  MoveC 1160 to (433.16, -30.09, -5) mm, rotated rx -180 ry 0 rz -60 deg; joints [3.301, -66.266, 153.274, -56.747, -88.159, 3.391] to (420.46, -17.39, -5) mm, rotated rx 180 ry 0 rz -60 deg; joints [4.068, -65.905, 152.306, -55.999, -87.786, 3.873]
  MoveL 1161 to (395.06, -17.39, -5) mm, rotated rx -180 ry 0 rz -30 deg; joints [13.007, -68.027, 157.856, -16.999, -89.219, 0.721]
  MoveL 1162 to (318.86, -17.39, -5) mm, rotated rx -180 ry 0 rz 0 deg; joints [22.894, -66.084, 152.119, 22.962, -85.478, -1.274]
  MoveC 1163 to (306.16, -30.09, -5) mm, rotated rx 180 ry 0 rz 0 deg; joints [21.838, -65.873, 151.62, 21.912, -85.183, -1.314] to (293.46, -17.39, -5) mm, rotated rx -180 ry 0 rz 0 deg; joints [22.278, -65.412, 150.426, 22.379, -84.518, -1.624]
  MoveL 1164 to (191.86, -17.39, -5) mm, rotated rx -180 ry 0 rz 0 deg; joints [20.102, -62.526, 143.489, 20.378, -80.65, -2.863]
  MoveC 1165 to (179.16, -30.09, -5) mm, rotated rx -180 ry 0 rz 0 deg; joints [19.189, -62.27, 142.918, 19.471, -80.304, -2.833] to (166.46, -17.39, -5) mm, rotated rx -180 ry 0 rz 0 deg; joints [19.62, -61.76, 141.713, 19.95, -79.673, -3.141]
  MoveL 1166 to (90.26, -17.39, -5) mm, rotated rx -180 ry 0 rz 0 deg; joints [18.3, -59.367, 136.274, 18.815, -76.713, -3.918]
  MoveL 1167 to (64.86, -17.39, -5) mm, rotated rx -180 ry 0 rz 0 deg; joints [17.897, -58.538, 134.424, 18.482, -75.714, -4.162]
  MoveC 1168 to (61.14, -26.37, -5) mm, rotated rx -180 ry 0 rz 0 deg; joints [17.408, -58.504, 134.36, 17.981, -75.65, -4.054] to (52.16, -30.09, -5) mm, rotated rx -180 ry 0 rz 0 deg; joints [17.095, -58.242, 133.784, 17.684, -75.327, -4.078]
  MoveL 1169 to (52.16, -30.09, -5) mm, rotated rx -180 ry 0 rz 0 deg; joints [17.095, -58.242, 133.784, 17.684, -75.327, -4.078]
  MoveC 1170 to (43.18, -26.37, -5) mm, rotated rx -180 ry 0 rz 0 deg; joints [17.141, -57.907, 133.035, 17.765, -74.936, -4.219] to (39.46, -17.39, -5) mm, rotated rx -180 ry 0 rz 0 deg; joints [17.511, -57.695, 132.553, 18.169, -74.709, -4.4]
  MoveL 1171 to (14.06, -17.39, -5) mm, rotated rx -180 ry 0 rz 0 deg; joints [17.141, -56.836, 130.661, 17.877, -73.696, -4.634]
  MoveC 1172 to (13.61, -17.2, -5) mm, rotated rx -180 ry 0 rz 0 deg; joints [17.143, -56.818, 130.623, 17.881, -73.676, -4.641] to (13.42, -16.75, -5) mm, rotated rx -180 ry 0 rz 0 deg; joints [17.161, -56.808, 130.599, 17.901, -73.665, -4.65]
  MoveL 1173 to (13.42, -16.12, -5) mm, rotated rx 180 ry 0 rz 0 deg; joints [17.191, -56.801, 130.584, 17.932, -73.659, -4.661]
  MoveC 1174 to (13.42, -15.67, -4.81) mm, rotated rx -180 ry 0 rz 0 deg; joints [17.211, -56.81, 130.574, 17.955, -73.643, -4.673] to (13.42, -15.48, -4.37) mm, rotated rx -180 ry 0 rz 0 deg; joints [17.22, -56.839, 130.571, 17.967, -73.613, -4.686]
  Set speed (500.0 mm/s)
  MoveL 1175 to (13.42, -15.48, 5) mm, rotated rx -180 ry 0 rz 0 deg; joints [17.216, -57.49, 130.588, 18.021, -73.01, -4.889]
  MoveL 1176 to (12.15, -16.75, 5) mm, rotated rx 180 ry 0 rz 0 deg; joints [17.139, -57.459, 130.522, 17.945, -72.97, -4.878]
  Set speed (25.4 mm/s)
  MoveL 1177 to (12.15, -16.75, 1) mm, rotated rx -180 ry 0 rz 0 deg; joints [17.141, -57.181, 130.516, 17.921, -73.228, -4.791]
  MoveL 1178 to (12.15, -16.75, -7.72) mm, rotated rx 180 ry 0 rz 0 deg; joints [17.144, -56.575, 130.497, 17.871, -73.788, -4.604]
  MoveC 1179 to (12.34, -16.75, -8.16) mm, rotated rx -180 ry 0 rz 0 deg; joints [17.147, -56.55, 130.51, 17.871, -73.824, -4.592] to (12.79, -16.75, -8.35) mm, rotated rx 180 ry 0 rz 0 deg; joints [17.154, -56.552, 130.543, 17.875, -73.854, -4.584]
  Set speed (50.8 mm/s)
  MoveL 1180 to (13.42, -16.75, -8.35) mm, rotated rx -180 ry 0 rz 0 deg; joints [17.163, -56.574, 130.591, 17.882, -73.88, -4.578]
  MoveC 1181 to (13.87, -16.94, -8.35) mm, rotated rx -180 ry 0 rz 0 deg; joints [17.161, -56.591, 130.628, 17.878, -73.899, -4.571] to (14.06, -17.39, -8.35) mm, rotated rx -180 ry 0 rz 0 deg; joints [17.143, -56.601, 130.653, 17.858, -73.911, -4.562]
  MoveL 1182 to (14.06, -169.79, -8.35) mm, rotated rx -180 ry 0 rz 0 deg; joints [9.848, -57.754, 133.422, 10.193, -75.015, -2.239]
  MoveL 1183 to (471.26, -169.79, -8.35) mm, rotated rx -180 ry 0 rz -60 deg; joints [-6.049, -66.719, 155.749, -66.059, -89.408, 1.775]
  MoveL 1184 to (471.26, -17.39, -8.35) mm, rotated rx 180 ry 0 rz -60 deg; joints [4.314, -66.857, 155.917, -55.696, -89.272, 1.665]
  MoveL 1185 to (445.86, -17.39, -8.35) mm, rotated rx -180 ry 0 rz -60 deg; joints [4.188, -66.217, 154.11, -55.84, -88.618, 2.632]
  MoveC 1186 to (433.16, -30.09, -8.35) mm, rotated rx -180 ry 0 rz -60 deg; joints [3.303, -65.899, 153.262, -56.737, -88.354, 3.094] to (420.46, -17.39, -8.35) mm, rotated rx 180 ry 0 rz -60 deg; joints [4.069, -65.548, 152.294, -55.987, -87.979, 3.586]
  MoveL 1187 to (395.06, -17.39, -8.35) mm, rotated rx 180 ry 0 rz -30 deg; joints [13.009, -67.611, 157.843, -16.996, -89.605, 0.603]
  MoveL 1188 to (318.86, -17.39, -8.35) mm, rotated rx 180 ry 0 rz 0 deg; joints [22.896, -65.729, 152.107, 22.954, -85.795, -1.139]
  MoveC 1189 to (306.16, -30.09, -8.35) mm, rotated rx -180 ry 0 rz 0 deg; joints [21.84, -65.522, 151.609, 21.904, -85.499, -1.187] to (293.46, -17.39, -8.35) mm, rotated rx -180 ry 0 rz 0 deg; joints [22.28, -65.07, 150.415, 22.369, -84.823, -1.498]
  MoveL 1190 to (191.86, -17.39, -8.35) mm, rotated rx -180 ry 0 rz 0 deg; joints [20.104, -62.233, 143.48, 20.364, -80.916, -2.763]
  MoveC 1191 to (179.16, -30.09, -8.35) mm, rotated rx 180 ry 0 rz 0 deg; joints [19.19, -61.98, 142.909, 19.457, -80.568, -2.738] to (166.46, -17.39, -8.35) mm, rotated rx -180 ry 0 rz 0 deg; joints [19.622, -61.477, 141.703, 19.935, -79.93, -3.046]
  MoveL 1192 to (90.26, -17.39, -8.35) mm, rotated rx -180 ry 0 rz 0 deg; joints [18.302, -59.111, 136.266, 18.798, -76.947, -3.836]
  MoveL 1193 to (64.86, -17.39, -8.35) mm, rotated rx -180 ry 0 rz 0 deg; joints [17.899, -58.29, 134.415, 18.465, -75.942, -4.084]
  MoveC 1194 to (61.14, -26.37, -8.35) mm, rotated rx -180 ry 0 rz 0 deg; joints [17.41, -58.255, 134.351, 17.964, -75.878, -3.978] to (52.16, -30.09, -8.35) mm, rotated rx -180 ry 0 rz 0 deg; joints [17.097, -57.996, 133.775, 17.667, -75.553, -4.004]
  MoveL 1195 to (52.16, -30.09, -8.35) mm, rotated rx -180 ry 0 rz 0 deg; joints [17.097, -57.996, 133.775, 17.667, -75.553, -4.004]
  MoveC 1196 to (43.18, -26.37, -8.35) mm, rotated rx -180 ry 0 rz 0 deg; joints [17.142, -57.664, 133.027, 17.747, -75.16, -4.146] to (39.46, -17.39, -8.35) mm, rotated rx -180 ry 0 rz 0 deg; joints [17.513, -57.453, 132.544, 18.151, -74.93, -4.325]
  MoveL 1197 to (14.06, -17.39, -8.35) mm, rotated rx -180 ry 0 rz 0 deg; joints [17.143, -56.601, 130.653, 17.858, -73.911, -4.562]
  MoveC 1198 to (13.61, -17.2, -8.35) mm, rotated rx -180 ry 0 rz 0 deg; joints [17.145, -56.584, 130.615, 17.862, -73.891, -4.569] to (13.42, -16.75, -8.35) mm, rotated rx -180 ry 0 rz 0 deg; joints [17.163, -56.574, 130.591, 17.882, -73.88, -4.578]
  MoveL 1199 to (13.42, -16.12, -8.35) mm, rotated rx -180 ry 0 rz 0 deg; joints [17.192, -56.567, 130.576, 17.913, -73.874, -4.589]
  MoveC 1200 to (13.42, -15.67, -8.16) mm, rotated rx -180 ry 0 rz 0 deg; joints [17.213, -56.576, 130.566, 17.936, -73.858, -4.601] to (13.42, -15.48, -7.72) mm, rotated rx -180 ry 0 rz 0 deg; joints [17.221, -56.606, 130.563, 17.948, -73.828, -4.613]
  Set speed (500.0 mm/s)
  MoveL 1201 to (13.42, -15.48, 6) mm, rotated rx -180 ry 0 rz 0 deg; joints [17.215, -57.56, 130.589, 18.027, -72.945, -4.911]
  MoveL 1202 to (-18.41, -15.48, 6) mm, rotated rx -180 ry 0 rz 0 deg; joints [16.771, -56.434, 128.187, 17.688, -71.688, -5.187]
  Set speed (25.4 mm/s)
  MoveL 1203 to (-18.41, -15.48, -4.37) mm, rotated rx -180 ry 0 rz 0 deg; joints [16.775, -55.739, 128.169, 17.626, -72.334, -4.973]
  MoveC 1204 to (-18.41, -15.67, -4.81) mm, rotated rx 180 ry 0 rz 0 deg; joints [16.767, -55.711, 128.173, 17.614, -72.363, -4.96] to (-18.41, -16.12, -5) mm, rotated rx -180 ry 0 rz 0 deg; joints [16.747, -55.703, 128.182, 17.591, -72.379, -4.948]
  Set speed (50.8 mm/s)
  MoveL 1205 to (-18.41, -16.75, -5) mm, rotated rx -180 ry 0 rz 0 deg; joints [16.718, -55.709, 128.197, 17.56, -72.384, -4.937]
  MoveC 1206 to (-18.6, -17.2, -5) mm, rotated rx 180 ry 0 rz 0 deg; joints [16.695, -55.707, 128.193, 17.537, -72.38, -4.931] to (-19.04, -17.39, -5) mm, rotated rx -180 ry 0 rz 0 deg; joints [16.681, -55.693, 128.163, 17.523, -72.364, -4.932]
  MoveL 1207 to (-39.46, -17.39, -5) mm, rotated rx -180 ry 0 rz 0 deg; joints [16.409, -54.976, 126.603, 17.321, -71.535, -5.113]
  MoveC 1208 to (-52.16, -30.09, -5) mm, rotated rx -180 ry 0 rz 0 deg; joints [15.682, -54.647, 125.906, 16.593, -71.115, -4.993] to (-64.86, -17.39, -5) mm, rotated rx -180 ry 0 rz 0 deg; joints [16.082, -54.069, 124.641, 17.084, -70.495, -5.336]
  MoveL 1209 to (-90.26, -17.39, -5) mm, rotated rx -180 ry 0 rz 0 deg; joints [15.768, -53.146, 122.653, 16.865, -69.445, -5.558]
  MoveL 1210 to (-166.46, -17.39, -5) mm, rotated rx 180 ry 0 rz 0 deg; joints [14.894, -50.279, 116.527, 16.305, -66.228, -6.221]
  MoveC 1211 to (-179.16, -30.09, -5) mm, rotated rx -180 ry 0 rz 0 deg; joints [14.242, -49.907, 115.751, 15.645, -65.767, -6.064] to (-191.86, -17.39, -5) mm, rotated rx -180 ry 0 rz 0 deg; joints [14.623, -49.288, 114.425, 16.15, -65.13, -6.444]
  MoveL 1212 to (-293.46, -17.39, -5) mm, rotated rx -180 ry 0 rz 0 deg; joints [13.63, -45.126, 105.665, 15.689, -60.583, -7.372]
  MoveC 1213 to (-306.16, -30.09, -5) mm, rotated rx -180 ry 0 rz 0 deg; joints [13.04, -44.706, 104.795, 15.083, -60.073, -7.184] to (-318.86, -17.39, -5) mm, rotated rx -180 ry 0 rz 0 deg; joints [13.402, -44.031, 103.374, 15.614, -59.402, -7.617]
  MoveL 1214 to (-395.06, -17.39, -5) mm, rotated rx -180 ry 0 rz 0 deg; joints [12.761, -40.591, 96.21, 15.497, -55.722, -8.407]
  MoveL 1215 to (-420.46, -17.39, -5) mm, rotated rx 180 ry 0 rz 0 deg; joints [12.56, -39.385, 93.71, 15.497, -54.444, -8.693]
  MoveC 1216 to (-433.16, -30.09, -5) mm, rotated rx 180 ry 0 rz 0 deg; joints [12.022, -38.9, 92.714, 14.938, -53.869, -8.482] to (-445.86, -17.39, -5) mm, rotated rx -180 ry 0 rz 0 deg; joints [12.366, -38.146, 91.146, 15.519, -53.136, -8.995]
  MoveL 1217 to (-471.26, -17.39, -5) mm, rotated rx -180 ry 0 rz 0 deg; joints [12.178, -36.871, 88.511, 15.564, -51.795, -9.314]
  MoveL 1218 to (-471.26, -169.79, -5) mm, rotated rx -180 ry 0 rz 0 deg; joints [6.925, -38.12, 91.194, 8.733, -52.522, -4.962]
  MoveL 1219 to (-14.06, -169.79, -5) mm, rotated rx -180 ry 0 rz 0 deg; joints [9.613, -57.027, 131.277, 10.019, -73.608, -2.435]
  MoveL 1220 to (-14.06, -17.39, -5) mm, rotated rx 180 ry 0 rz 0 deg; joints [16.749, -55.867, 128.542, 17.574, -72.565, -4.887]
  MoveL 1221 to (-19.04, -17.39, -5) mm, rotated rx -180 ry 0 rz 0 deg; joints [16.681, -55.693, 128.163, 17.523, -72.364, -4.932]
  MoveC 1222 to (-19.49, -17.2, -5) mm, rotated rx -180 ry 0 rz 0 deg; joints [16.683, -55.676, 128.125, 17.528, -72.344, -4.939] to (-19.68, -16.75, -5) mm, rotated rx -180 ry 0 rz 0 deg; joints [16.701, -55.665, 128.1, 17.547, -72.333, -4.949]
  MoveL 1223 to (-19.68, -16.12, -5) mm, rotated rx -180 ry 0 rz 0 deg; joints [16.73, -55.659, 128.086, 17.578, -72.327, -4.96]
  MoveC 1224 to (-19.68, -15.67, -4.81) mm, rotated rx -180 ry 0 rz 0 deg; joints [16.75, -55.667, 128.076, 17.601, -72.312, -4.972] to (-19.68, -15.48, -4.37) mm, rotated rx 180 ry 0 rz 0 deg; joints [16.758, -55.695, 128.073, 17.613, -72.283, -4.984]
  Set speed (500.0 mm/s)
  MoveL 1225 to (-19.68, -15.48, 5) mm, rotated rx 180 ry 0 rz 0 deg; joints [16.754, -56.322, 128.089, 17.669, -71.7, -5.178]
  MoveL 1226 to (-18.41, -15.48, 5) mm, rotated rx -180 ry 0 rz 0 deg; joints [16.771, -56.368, 128.186, 17.682, -71.751, -5.167]
  Set speed (25.4 mm/s)
  MoveL 1227 to (-18.41, -15.48, 1) mm, rotated rx -180 ry 0 rz 0 deg; joints [16.773, -56.1, 128.18, 17.657, -72.001, -5.083]
  MoveL 1228 to (-18.41, -15.48, -7.72) mm, rotated rx -180 ry 0 rz 0 deg; joints [16.777, -55.514, 128.161, 17.606, -72.542, -4.904]
  MoveC 1229 to (-18.41, -15.67, -8.16) mm, rotated rx -180 ry 0 rz 0 deg; joints [16.769, -55.485, 128.164, 17.595, -72.571, -4.892] to (-18.41, -16.12, -8.35) mm, rotated rx -180 ry 0 rz 0 deg; joints [16.748, -55.477, 128.174, 17.572, -72.586, -4.88]
  Set speed (50.8 mm/s)
  MoveL 1230 to (-18.41, -16.75, -8.35) mm, rotated rx -180 ry 0 rz 0 deg; joints [16.72, -55.483, 128.189, 17.541, -72.592, -4.869]
  MoveC 1231 to (-18.6, -17.2, -8.35) mm, rotated rx 180 ry 0 rz 0 deg; joints [16.697, -55.481, 128.185, 17.518, -72.588, -4.863] to (-19.04, -17.39, -8.35) mm, rotated rx -180 ry 0 rz 0 deg; joints [16.682, -55.468, 128.155, 17.504, -72.571, -4.863]
  MoveL 1232 to (-39.46, -17.39, -8.35) mm, rotated rx 180 ry 0 rz 0 deg; joints [16.41, -54.755, 126.595, 17.301, -71.738, -5.047]
  MoveC 1233 to (-52.16, -30.09, -8.35) mm, rotated rx -180 ry 0 rz 0 deg; joints [15.683, -54.428, 125.898, 16.574, -71.317, -4.929] to (-64.86, -17.39, -8.35) mm, rotated rx -180 ry 0 rz 0 deg; joints [16.084, -53.854, 124.633, 17.064, -70.693, -5.272]
  MoveL 1234 to (-90.26, -17.39, -8.35) mm, rotated rx -180 ry 0 rz 0 deg; joints [15.769, -52.937, 122.646, 16.844, -69.638, -5.496]
  MoveL 1235 to (-166.46, -17.39, -8.35) mm, rotated rx -180 ry 0 rz 0 deg; joints [14.895, -50.085, 116.519, 16.283, -66.407, -6.165]
  MoveC 1236 to (-179.16, -30.09, -8.35) mm, rotated rx 180 ry 0 rz 0 deg; joints [14.243, -49.715, 115.744, 15.624, -65.945, -6.01] to (-191.86, -17.39, -8.35) mm, rotated rx -180 ry 0 rz 0 deg; joints [14.624, -49.098, 114.417, 16.128, -65.305, -6.389]
  MoveL 1237 to (-293.46, -17.39, -8.35) mm, rotated rx 180 ry 0 rz 0 deg; joints [13.631, -44.953, 105.657, 15.665, -60.743, -7.321]
  MoveC 1238 to (-306.16, -30.09, -8.35) mm, rotated rx -180 ry 0 rz 0 deg; joints [13.041, -44.534, 104.788, 15.06, -60.232, -7.135] to (-318.86, -17.39, -8.35) mm, rotated rx -180 ry 0 rz 0 deg; joints [13.403, -43.862, 103.367, 15.59, -59.558, -7.567]
  MoveL 1239 to (-395.06, -17.39, -8.35) mm, rotated rx -180 ry 0 rz 0 deg; joints [12.762, -40.431, 96.203, 15.471, -55.869, -8.358]
  MoveL 1240 to (-420.46, -17.39, -8.35) mm, rotated rx 180 ry 0 rz 0 deg; joints [12.561, -39.229, 93.703, 15.47, -54.588, -8.645]
  MoveC 1241 to (-433.16, -30.09, -8.35) mm, rotated rx -180 ry 0 rz 0 deg; joints [12.023, -38.744, 92.707, 14.911, -54.012, -8.436] to (-445.86, -17.39, -8.35) mm, rotated rx -180 ry 0 rz 0 deg; joints [12.367, -37.993, 91.139, 15.491, -53.277, -8.947]
  MoveL 1242 to (-471.26, -17.39, -8.35) mm, rotated rx 180 ry 0 rz 0 deg; joints [12.178, -36.721, 88.504, 15.535, -51.933, -9.266]
  MoveL 1243 to (-471.26, -169.79, -8.35) mm, rotated rx 180 ry 0 rz 0 deg; joints [6.926, -37.966, 91.187, 8.717, -52.667, -4.934]
  MoveL 1244 to (-14.06, -169.79, -8.35) mm, rotated rx -180 ry 0 rz 0 deg; joints [9.614, -56.791, 131.269, 10.008, -73.832, -2.394]
  MoveL 1245 to (-14.06, -17.39, -8.35) mm, rotated rx -180 ry 0 rz 0 deg; joints [16.75, -55.64, 128.534, 17.555, -72.774, -4.818]
  MoveL 1246 to (-19.04, -17.39, -8.35) mm, rotated rx -180 ry 0 rz 0 deg; joints [16.682, -55.468, 128.155, 17.504, -72.571, -4.863]
  MoveC 1247 to (-19.49, -17.2, -8.35) mm, rotated rx -180 ry 0 rz 0 deg; joints [16.685, -55.45, 128.117, 17.508, -72.551, -4.871] to (-19.68, -16.75, -8.35) mm, rotated rx -180 ry 0 rz 0 deg; joints [16.702, -55.439, 128.092, 17.528, -72.54, -4.88]
  MoveL 1248 to (-19.68, -16.12, -8.35) mm, rotated rx -180 ry 0 rz 0 deg; joints [16.731, -55.433, 128.078, 17.559, -72.535, -4.891]
  MoveC 1249 to (-19.68, -15.67, -8.16) mm, rotated rx -180 ry 0 rz 0 deg; joints [16.751, -55.441, 128.068, 17.582, -72.519, -4.903] to (-19.68, -15.48, -7.72) mm, rotated rx -180 ry 0 rz 0 deg; joints [16.76, -55.47, 128.065, 17.593, -72.49, -4.916]
  Set speed (500.0 mm/s)
  MoveL 1250 to (-19.68, -15.48, 6) mm, rotated rx 180 ry 0 rz 0 deg; joints [16.754, -56.389, 128.091, 17.675, -71.638, -5.198]
  MoveL 1251 to (-13.42, -196.52, 6) mm, rotated rx 180 ry 0 rz 0 deg; joints [8.324, -57.961, 131.671, 8.701, -73.018, -2.16]
  Set speed (25.4 mm/s)
  MoveL 1252 to (-13.42, -196.51, -4.36) mm, rotated rx -180 ry 0 rz 0 deg; joints [8.327, -57.228, 131.652, 8.672, -73.724, -2.048]
  MoveC 1253 to (-13.42, -196.7, -4.81) mm, rotated rx -180 ry 0 rz 0 deg; joints [8.318, -57.197, 131.653, 8.661, -73.755, -2.041] to (-13.42, -197.15, -5) mm, rotated rx 180 ry 0 rz 0 deg; joints [8.297, -57.186, 131.658, 8.638, -73.77, -2.032]
  Set speed (50.8 mm/s)
  MoveL 1254 to (-13.42, -197.79, -5) mm, rotated rx 180 ry 0 rz 0 deg; joints [8.266, -57.189, 131.665, 8.606, -73.773, -2.023]
  MoveC 1255 to (-13.61, -198.23, -5) mm, rotated rx -180 ry 0 rz 0 deg; joints [8.243, -57.184, 131.656, 8.582, -73.767, -2.018] to (-14.06, -198.42, -5) mm, rotated rx -180 ry 0 rz 0 deg; joints [8.23, -57.17, 131.623, 8.57, -73.749, -2.017]
  MoveL 1256 to (-39.46, -198.42, -5) mm, rotated rx 180 ry 0 rz 0 deg; joints [8.056, -56.276, 129.652, 8.437, -72.676, -2.133]
  MoveC 1257 to (-52.16, -211.12, -5) mm, rotated rx -180 ry 0 rz 0 deg; joints [7.375, -55.879, 128.793, 7.743, -72.191, -1.996] to (-64.86, -198.42, -5) mm, rotated rx -180 ry 0 rz 0 deg; joints [7.889, -55.367, 127.661, 8.312, -71.598, -2.248]
  MoveL 1258 to (-90.26, -198.42, -5) mm, rotated rx -180 ry 0 rz 0 deg; joints [7.729, -54.442, 125.647, 8.197, -70.513, -2.361]
  MoveL 1259 to (-166.46, -198.42, -5) mm, rotated rx -180 ry 0 rz 0 deg; joints [7.285, -51.573, 119.46, 7.9, -67.207, -2.694]
  MoveC 1260 to (-179.16, -211.12, -5) mm, rotated rx 180 ry 0 rz 0 deg; joints [6.674, -51.136, 118.535, 7.265, -66.692, -2.514] to (-191.86, -198.42, -5) mm, rotated rx -180 ry 0 rz 0 deg; joints [7.148, -50.583, 117.344, 7.818, -66.084, -2.805]
  MoveL 1261 to (-293.46, -198.42, -5) mm, rotated rx -180 ry 0 rz 0 deg; joints [6.648, -46.437, 108.562, 7.567, -61.46, -3.258]
  MoveC 1262 to (-306.16, -211.12, -5) mm, rotated rx 180 ry 0 rz 0 deg; joints [6.095, -45.951, 107.55, 6.973, -60.905, -3.039] to (-318.86, -198.42, -5) mm, rotated rx 180 ry 0 rz 0 deg; joints [6.534, -45.349, 106.274, 7.524, -60.264, -3.376]
  MoveL 1263 to (-395.06, -198.42, -5) mm, rotated rx -180 ry 0 rz 0 deg; joints [6.213, -41.939, 99.145, 7.446, -56.555, -3.753]
  MoveL 1264 to (-420.46, -198.42, -5) mm, rotated rx -180 ry 0 rz 0 deg; joints [6.113, -40.749, 96.667, 7.439, -55.271, -3.889]
  MoveC 1265 to (-433.16, -211.12, -5) mm, rotated rx 180 ry 0 rz 0 deg; joints [5.608, -40.201, 95.535, 6.874, -54.656, -3.632] to (-445.86, -198.42, -5) mm, rotated rx -180 ry 0 rz 0 deg; joints [6.016, -39.527, 94.13, 7.441, -53.959, -4.031]
  MoveL 1266 to (-471.26, -198.42, -5) mm, rotated rx 180 ry 0 rz 0 deg; joints [5.922, -38.273, 91.528, 7.455, -52.616, -4.18]
  MoveL 1267 to (-471.26, -350.82, -5) mm, rotated rx 180 ry 0 rz 0 deg; joints [0.538, -38.663, 92.418, 0.669, -52.887, -0.124]
  MoveL 1268 to (-14.06, -350.82, -5) mm, rotated rx 180 ry 0 rz 0 deg; joints [0.749, -57.524, 132.551, 0.774, -74.159, 0.072]
  MoveL 1269 to (-14.06, -198.42, -5) mm, rotated rx -180 ry 0 rz 0 deg; joints [8.23, -57.17, 131.623, 8.57, -73.749, -2.017]
  MoveC 1270 to (-13.87, -197.97, -5) mm, rotated rx 180 ry 0 rz 0 deg; joints [8.254, -57.174, 131.633, 8.594, -73.755, -2.023] to (-13.42, -197.79, -5) mm, rotated rx 180 ry 0 rz 0 deg; joints [8.266, -57.189, 131.665, 8.606, -73.773, -2.023]
  MoveL 1271 to (-12.79, -197.79, -5) mm, rotated rx 180 ry 0 rz 0 deg; joints [8.27, -57.211, 131.714, 8.609, -73.799, -2.02]
  MoveC 1272 to (-12.34, -197.79, -4.81) mm, rotated rx 180 ry 0 rz 0 deg; joints [8.273, -57.24, 131.749, 8.612, -73.806, -2.02] to (-12.15, -197.78, -4.37) mm, rotated rx -180 ry 0 rz 0 deg; joints [8.274, -57.278, 131.765, 8.615, -73.783, -2.024]
  Set speed (500.0 mm/s)
  MoveL 1273 to (-12.15, -197.79, 5) mm, rotated rx 180 ry 0 rz 0 deg; joints [8.271, -57.941, 131.782, 8.64, -73.145, -2.124]
  MoveL 1274 to (-13.42, -196.52, 5) mm, rotated rx 180 ry 0 rz 0 deg; joints [8.324, -57.89, 131.67, 8.698, -73.087, -2.149]
  Set speed (25.4 mm/s)
  MoveL 1275 to (-13.42, -196.51, 1) mm, rotated rx 180 ry 0 rz 0 deg; joints [8.325, -57.608, 131.664, 8.687, -73.359, -2.106]
  MoveL 1276 to (-13.42, -196.52, -7.72) mm, rotated rx -180 ry 0 rz 0 deg; joints [8.328, -56.99, 131.644, 8.663, -73.951, -2.013]
  MoveC 1277 to (-13.42, -196.7, -8.16) mm, rotated rx 180 ry 0 rz 0 deg; joints [8.319, -56.959, 131.645, 8.653, -73.982, -2.005] to (-13.42, -197.15, -8.35) mm, rotated rx -180 ry 0 rz 0 deg; joints [8.298, -56.948, 131.65, 8.629, -73.996, -1.997]
  Set speed (50.8 mm/s)
  MoveL 1278 to (-13.42, -197.79, -8.35) mm, rotated rx -180 ry 0 rz 0 deg; joints [8.267, -56.951, 131.657, 8.597, -73.999, -1.988]
  MoveC 1279 to (-13.61, -198.23, -8.35) mm, rotated rx 180 ry 0 rz 0 deg; joints [8.244, -56.947, 131.647, 8.573, -73.994, -1.982] to (-14.06, -198.42, -8.35) mm, rotated rx -180 ry 0 rz 0 deg; joints [8.232, -56.932, 131.615, 8.562, -73.975, -1.982]
  MoveL 1280 to (-39.46, -198.42, -8.35) mm, rotated rx 180 ry 0 rz 0 deg; joints [8.057, -56.045, 129.644, 8.428, -72.896, -2.1]
  MoveC 1281 to (-52.16, -211.12, -8.35) mm, rotated rx -180 ry 0 rz 0 deg; joints [7.376, -55.651, 128.785, 7.734, -72.409, -1.966] to (-64.86, -198.42, -8.35) mm, rotated rx -180 ry 0 rz 0 deg; joints [7.89, -55.143, 127.653, 8.303, -71.812, -2.215]
  MoveL 1282 to (-90.26, -198.42, -8.35) mm, rotated rx -180 ry 0 rz 0 deg; joints [7.73, -54.224, 125.639, 8.187, -70.721, -2.329]
  MoveL 1283 to (-166.46, -198.42, -8.35) mm, rotated rx -180 ry 0 rz 0 deg; joints [7.286, -51.372, 119.453, 7.89, -67.398, -2.665]
  MoveC 1284 to (-179.16, -211.12, -8.35) mm, rotated rx -180 ry 0 rz 0 deg; joints [6.675, -50.937, 118.527, 7.255, -66.882, -2.488] to (-191.86, -198.42, -8.35) mm, rotated rx 180 ry 0 rz 0 deg; joints [7.149, -50.387, 117.337, 7.808, -66.271, -2.777]
  MoveL 1285 to (-293.46, -198.42, -8.35) mm, rotated rx 180 ry 0 rz 0 deg; joints [6.649, -46.258, 108.554, 7.556, -61.63, -3.233]
  MoveC 1286 to (-306.16, -211.12, -8.35) mm, rotated rx 180 ry 0 rz 0 deg; joints [6.095, -45.775, 107.542, 6.963, -61.073, -3.016] to (-318.86, -198.42, -8.35) mm, rotated rx -180 ry 0 rz 0 deg; joints [6.534, -45.174, 106.267, 7.513, -60.43, -3.352]
  MoveL 1287 to (-395.06, -198.42, -8.35) mm, rotated rx -180 ry 0 rz 0 deg; joints [6.214, -41.776, 99.138, 7.434, -56.71, -3.73]
  MoveL 1288 to (-420.46, -198.42, -8.35) mm, rotated rx -180 ry 0 rz 0 deg; joints [6.114, -40.588, 96.659, 7.426, -55.422, -3.865]
  MoveC 1289 to (-433.16, -211.12, -8.35) mm, rotated rx -180 ry 0 rz 0 deg; joints [5.608, -40.042, 95.528, 6.862, -54.807, -3.61] to (-445.86, -198.42, -8.35) mm, rotated rx -180 ry 0 rz 0 deg; joints [6.017, -39.37, 94.122, 7.428, -54.107, -4.007]
  MoveL 1290 to (-471.26, -198.42, -8.35) mm, rotated rx -180 ry 0 rz 0 deg; joints [5.923, -38.119, 91.521, 7.441, -52.762, -4.157]
  MoveL 1291 to (-471.26, -350.82, -8.35) mm, rotated rx -180 ry 0 rz 0 deg; joints [0.539, -38.508, 92.411, 0.669, -53.035, -0.122]
  MoveL 1292 to (-14.06, -350.82, -8.35) mm, rotated rx -180 ry 0 rz 0 deg; joints [0.75, -57.282, 132.542, 0.774, -74.391, 0.075]
  MoveL 1293 to (-14.06, -198.42, -8.35) mm, rotated rx -180 ry 0 rz 0 deg; joints [8.232, -56.932, 131.615, 8.562, -73.975, -1.982]
  MoveC 1294 to (-13.87, -197.97, -8.35) mm, rotated rx 180 ry 0 rz 0 deg; joints [8.255, -56.936, 131.624, 8.585, -73.981, -1.987] to (-13.42, -197.79, -8.35) mm, rotated rx -180 ry 0 rz 0 deg; joints [8.267, -56.951, 131.657, 8.597, -73.999, -1.988]
  MoveL 1295 to (-12.79, -197.78, -8.35) mm, rotated rx -180 ry 0 rz 0 deg; joints [8.271, -56.973, 131.706, 8.601, -74.026, -1.985]
  MoveC 1296 to (-12.34, -197.78, -8.16) mm, rotated rx 180 ry 0 rz 0 deg; joints [8.274, -57.002, 131.741, 8.604, -74.033, -1.985] to (-12.15, -197.79, -7.72) mm, rotated rx -180 ry 0 rz 0 deg; joints [8.276, -57.04, 131.756, 8.606, -74.01, -1.988]
  Set speed (500.0 mm/s)
  MoveL 1297 to (-12.15, -197.79, 6) mm, rotated rx 180 ry 0 rz 0 deg; joints [8.271, -58.012, 131.784, 8.643, -73.076, -2.135]
  MoveL 1298 to (12.15, -197.78, 6) mm, rotated rx -180 ry 0 rz 0 deg; joints [8.446, -58.875, 133.65, 8.78, -74.075, -2.025]
  Set speed (25.4 mm/s)
  MoveL 1299 to (12.15, -197.79, -4.36) mm, rotated rx 180 ry 0 rz 0 deg; joints [8.449, -58.119, 133.631, 8.753, -74.803, -1.91]
  MoveC 1300 to (12.34, -197.79, -4.81) mm, rotated rx -180 ry 0 rz 0 deg; joints [8.451, -58.093, 133.644, 8.753, -74.842, -1.904] to (12.79, -197.78, -5) mm, rotated rx -180 ry 0 rz 0 deg; joints [8.454, -58.095, 133.677, 8.755, -74.874, -1.9]
  Set speed (50.8 mm/s)
  MoveL 1301 to (13.42, -197.78, -5) mm, rotated rx -180 ry 0 rz 0 deg; joints [8.459, -58.117, 133.726, 8.759, -74.9, -1.897]
  MoveC 1302 to (13.87, -197.97, -5) mm, rotated rx -180 ry 0 rz 0 deg; joints [8.453, -58.133, 133.762, 8.752, -74.92, -1.892] to (14.06, -198.42, -5) mm, rotated rx -180 ry 0 rz 0 deg; joints [8.432, -58.141, 133.782, 8.73, -74.93, -1.885]
  MoveL 1303 to (14.06, -350.82, -5) mm, rotated rx -180 ry 0 rz 0 deg; joints [0.767, -58.495, 134.722, 0.789, -75.359, 0.085]
  MoveL 1304 to (471.26, -350.82, -5) mm, rotated rx -180 ry 0 rz -60 deg; joints [-17.82, -66.092, 153.07, -77.85, -89.164, 3.843]
  MoveL 1305 to (471.26, -198.42, -5) mm, rotated rx 180 ry 0 rz -60 deg; joints [-7.973, -67.012, 155.513, -67.988, -89.239, 2.279]
  MoveL 1306 to (445.86, -198.42, -5) mm, rotated rx -180 ry 0 rz -60 deg; joints [-7.742, -66.355, 153.715, -67.775, -88.802, 3.333]
  MoveC 1307 to (433.16, -211.12, -5) mm, rotated rx -180 ry 0 rz -60 deg; joints [-8.443, -65.964, 152.685, -68.49, -88.597, 3.94] to (420.46, -198.42, -5) mm, rotated rx -180 ry 0 rz -60 deg; joints [-7.523, -65.671, 151.907, -67.583, -88.364, 4.368]
  MoveL 1308 to (395.06, -198.42, -5) mm, rotated rx -180 ry 0 rz -60 deg; joints [-7.317, -64.963, 150.088, -67.41, -87.924, 5.389]
  MoveL 1309 to (318.86, -198.42, -5) mm, rotated rx 180 ry 0 rz 0 deg; joints [11.472, -67.344, 155.959, 11.476, -87.773, -0.003]
  MoveC 1310 to (306.16, -211.12, -5) mm, rotated rx 180 ry 0 rz 0 deg; joints [10.466, -67.073, 155.242, 10.472, -87.33, -0.06] to (293.46, -198.42, -5) mm, rotated rx 180 ry 0 rz 0 deg; joints [11.139, -66.691, 154.181, 11.152, -86.668, -0.213]
  MoveL 1311 to (191.86, -198.42, -5) mm, rotated rx -180 ry 0 rz 0 deg; joints [9.976, -63.84, 146.957, 10.061, -82.351, -0.928]
  MoveC 1312 to (179.16, -211.12, -5) mm, rotated rx -180 ry 0 rz 0 deg; joints [9.114, -63.516, 146.193, 9.202, -81.9, -0.896] to (166.46, -198.42, -5) mm, rotated rx -180 ry 0 rz 0 deg; joints [9.722, -63.077, 145.119, 9.832, -81.288, -1.082]
  MoveL 1313 to (90.26, -198.42, -5) mm, rotated rx -180 ry 0 rz 0 deg; joints [9.032, -60.681, 139.522, 9.226, -78.112, -1.506]
  MoveL 1314 to (64.86, -198.42, -5) mm, rotated rx 180 ry 0 rz 0 deg; joints [8.823, -59.85, 137.625, 9.049, -77.053, -1.636]
  MoveC 1315 to (61.14, -207.4, -5) mm, rotated rx -180 ry 0 rz 0 deg; joints [8.328, -59.766, 137.448, 8.546, -76.944, -1.545] to (52.16, -211.12, -5) mm, rotated rx 180 ry 0 rz 0 deg; joints [8.07, -59.484, 136.812, 8.292, -76.586, -1.541]
  MoveL 1316 to (52.16, -211.12, -5) mm, rotated rx 180 ry 0 rz 0 deg; joints [8.07, -59.484, 136.812, 8.292, -76.586, -1.541]
  MoveC 1317 to (43.18, -207.4, -5) mm, rotated rx -180 ry 0 rz 0 deg; joints [8.194, -59.168, 136.094, 8.435, -76.193, -1.629] to (39.46, -198.42, -5) mm, rotated rx 180 ry 0 rz 0 deg; joints [8.623, -59.003, 135.712, 8.884, -75.993, -1.763]
  MoveL 1318 to (14.06, -198.42, -5) mm, rotated rx -180 ry 0 rz 0 deg; joints [8.432, -58.141, 133.782, 8.73, -74.93, -1.885]
  MoveC 1319 to (13.61, -198.23, -5) mm, rotated rx -180 ry 0 rz 0 deg; joints [8.438, -58.125, 133.745, 8.736, -74.91, -1.89] to (13.42, -197.78, -5) mm, rotated rx -180 ry 0 rz 0 deg; joints [8.459, -58.117, 133.726, 8.759, -74.9, -1.897]
  MoveL 1320 to (13.42, -197.15, -5) mm, rotated rx -180 ry 0 rz 0 deg; joints [8.49, -58.114, 133.719, 8.791, -74.897, -1.905]
  MoveC 1321 to (13.42, -196.7, -4.81) mm, rotated rx -180 ry 0 rz 0 deg; joints [8.513, -58.125, 133.714, 8.815, -74.882, -1.914] to (13.42, -196.52, -4.37) mm, rotated rx 180 ry 0 rz 0 deg; joints [8.522, -58.157, 133.713, 8.826, -74.85, -1.921]
  Set speed (500.0 mm/s)
  MoveL 1322 to (13.42, -196.51, 5) mm, rotated rx -180 ry 0 rz 0 deg; joints [8.518, -58.841, 133.731, 8.851, -74.191, -2.027]
  MoveL 1323 to (12.15, -197.78, 5) mm, rotated rx -180 ry 0 rz 0 deg; joints [8.446, -58.803, 133.649, 8.777, -74.145, -2.014]
  Set speed (25.4 mm/s)
  MoveL 1324 to (12.15, -197.78, 1) mm, rotated rx 180 ry 0 rz 0 deg; joints [8.448, -58.511, 133.642, 8.767, -74.427, -1.969]
  MoveL 1325 to (12.15, -197.79, -7.72) mm, rotated rx -180 ry 0 rz 0 deg; joints [8.451, -57.874, 133.622, 8.744, -75.037, -1.873]
  MoveC 1326 to (12.34, -197.79, -8.16) mm, rotated rx 180 ry 0 rz 0 deg; joints [8.452, -57.848, 133.635, 8.744, -75.076, -1.867] to (12.79, -197.79, -8.35) mm, rotated rx 180 ry 0 rz 0 deg; joints [8.455, -57.849, 133.669, 8.746, -75.108, -1.863]
  Set speed (50.8 mm/s)
  MoveL 1327 to (13.42, -197.78, -8.35) mm, rotated rx -180 ry 0 rz 0 deg; joints [8.46, -57.871, 133.717, 8.75, -75.135, -1.86]
  MoveC 1328 to (13.87, -197.97, -8.35) mm, rotated rx 180 ry 0 rz 0 deg; joints [8.454, -57.887, 133.754, 8.743, -75.154, -1.855] to (14.06, -198.42, -8.35) mm, rotated rx 180 ry 0 rz 0 deg; joints [8.433, -57.895, 133.773, 8.721, -75.164, -1.848]
  MoveL 1329 to (14.06, -350.82, -8.35) mm, rotated rx 180 ry 0 rz 0 deg; joints [0.768, -58.245, 134.713, 0.789, -75.6, 0.088]
  MoveL 1330 to (471.26, -350.82, -8.35) mm, rotated rx -180 ry 0 rz -60 deg; joints [-17.82, -65.727, 153.058, -77.845, -89.239, 3.498]
  MoveL 1331 to (471.26, -198.42, -8.35) mm, rotated rx -180 ry 0 rz -60 deg; joints [-7.972, -66.622, 155.5, -67.983, -89.38, 1.93]
  MoveL 1332 to (445.86, -198.42, -8.35) mm, rotated rx -180 ry 0 rz -60 deg; joints [-7.741, -65.984, 153.703, -67.768, -88.937, 3.001]
  MoveC 1333 to (433.16, -211.12, -8.35) mm, rotated rx 180 ry 0 rz -60 deg; joints [-8.443, -65.603, 152.673, -68.481, -88.725, 3.615] to (420.46, -198.42, -8.35) mm, rotated rx 180 ry 0 rz -60 deg; joints [-7.523, -65.317, 151.895, -67.574, -88.494, 4.052]
  MoveL 1334 to (395.06, -198.42, -8.35) mm, rotated rx 180 ry 0 rz -60 deg; joints [-7.317, -64.624, 150.077, -67.399, -88.05, 5.087]
  MoveL 1335 to (318.86, -198.42, -8.35) mm, rotated rx -180 ry 0 rz 0 deg; joints [11.474, -66.95, 155.946, 11.475, -88.147, 0.073]
  MoveC 1336 to (306.16, -211.12, -8.35) mm, rotated rx -180 ry 0 rz 0 deg; joints [10.468, -66.686, 155.229, 10.471, -87.698, 0.008] to (293.46, -198.42, -8.35) mm, rotated rx 180 ry 0 rz 0 deg; joints [11.14, -66.316, 154.169, 11.15, -87.024, -0.143]
  MoveL 1337 to (191.86, -198.42, -8.35) mm, rotated rx -180 ry 0 rz 0 deg; joints [9.978, -63.525, 146.946, 10.056, -82.651, -0.874]
  MoveC 1338 to (179.16, -211.12, -8.35) mm, rotated rx -180 ry 0 rz 0 deg; joints [9.116, -63.206, 146.182, 9.196, -82.196, -0.848] to (166.46, -198.42, -8.35) mm, rotated rx -180 ry 0 rz 0 deg; joints [9.724, -62.774, 145.109, 9.825, -81.577, -1.032]
  MoveL 1339 to (90.26, -198.42, -8.35) mm, rotated rx -180 ry 0 rz 0 deg; joints [9.033, -60.409, 139.512, 9.219, -78.371, -1.463]
  MoveL 1340 to (64.86, -198.42, -8.35) mm, rotated rx -180 ry 0 rz 0 deg; joints [8.824, -59.587, 137.616, 9.042, -77.304, -1.596]
  MoveC 1341 to (61.14, -207.4, -8.35) mm, rotated rx 180 ry 0 rz 0 deg; joints [8.33, -59.505, 137.438, 8.538, -77.194, -1.506] to (52.16, -211.12, -8.35) mm, rotated rx 180 ry 0 rz 0 deg; joints [8.071, -59.225, 136.803, 8.285, -76.834, -1.504]
  MoveL 1342 to (52.16, -211.12, -8.35) mm, rotated rx 180 ry 0 rz 0 deg; joints [8.071, -59.225, 136.803, 8.285, -76.834, -1.504]
  MoveC 1343 to (43.18, -207.4, -8.35) mm, rotated rx 180 ry 0 rz 0 deg; joints [8.196, -58.912, 136.085, 8.427, -76.437, -1.592] to (39.46, -198.42, -8.35) mm, rotated rx -180 ry 0 rz 0 deg; joints [8.624, -58.749, 135.703, 8.876, -76.235, -1.724]
  MoveL 1344 to (14.06, -198.42, -8.35) mm, rotated rx 180 ry 0 rz 0 deg; joints [8.433, -57.895, 133.773, 8.721, -75.164, -1.848]
  MoveC 1345 to (13.61, -198.23, -8.35) mm, rotated rx 180 ry 0 rz 0 deg; joints [8.439, -57.879, 133.737, 8.728, -75.145, -1.853] to (13.42, -197.78, -8.35) mm, rotated rx -180 ry 0 rz 0 deg; joints [8.46, -57.871, 133.717, 8.75, -75.135, -1.86]
  MoveL 1346 to (13.42, -197.15, -8.35) mm, rotated rx -180 ry 0 rz 0 deg; joints [8.492, -57.868, 133.71, 8.783, -75.131, -1.868]
  MoveC 1347 to (13.42, -196.7, -8.16) mm, rotated rx 180 ry 0 rz 0 deg; joints [8.514, -57.88, 133.705, 8.806, -75.116, -1.876] to (13.42, -196.52, -7.72) mm, rotated rx -180 ry 0 rz 0 deg; joints [8.523, -57.912, 133.705, 8.817, -75.084, -1.884]
  Set speed (500.0 mm/s)
  MoveL 1348 to (13.42, -196.51, 6) mm, rotated rx 180 ry 0 rz 0 deg; joints [8.518, -58.914, 133.733, 8.853, -74.121, -2.038]
  MoveL 1349 to (12.15, -384.12, 6) mm, rotated rx -180 ry 0 rz 0 deg; joints [-0.922, -59.231, 134.593, -0.961, -74.494, 0.515]
  Set speed (25.4 mm/s)
  MoveL 1350 to (12.15, -384.12, -4.36) mm, rotated rx 180 ry 0 rz 0 deg; joints [-0.92, -58.464, 134.573, -0.955, -75.242, 0.502]
  MoveC 1351 to (12.34, -384.12, -4.81) mm, rotated rx -180 ry 0 rz 0 deg; joints [-0.92, -58.437, 134.586, -0.955, -75.282, 0.501] to (12.79, -384.12, -5) mm, rotated rx -180 ry 0 rz 0 deg; joints [-0.92, -58.438, 134.62, -0.955, -75.315, 0.501]
  Set speed (50.8 mm/s)
  MoveL 1352 to (13.42, -384.12, -5) mm, rotated rx 180 ry 0 rz 0 deg; joints [-0.921, -58.46, 134.669, -0.956, -75.342, 0.5]
  MoveC 1353 to (13.87, -384.31, -5) mm, rotated rx -180 ry 0 rz 0 deg; joints [-0.93, -58.475, 134.704, -0.966, -75.361, 0.502] to (14.06, -384.76, -5) mm, rotated rx -180 ry 0 rz 0 deg; joints [-0.953, -58.481, 134.717, -0.989, -75.369, 0.508]
  MoveL 1354 to (14.06, -537.16, -5) mm, rotated rx -180 ry 0 rz 0 deg; joints [-8.614, -58.004, 133.734, -8.923, -75.025, 2.464]
  MoveL 1355 to (471.26, -537.16, -5) mm, rotated rx -180 ry 0 rz -60 deg; joints [-28.512, -64.029, 147.744, -88.547, -89.64, 7.172]
  MoveL 1356 to (471.26, -384.76, -5) mm, rotated rx -180 ry 0 rz -60 deg; joints [-19.892, -65.794, 152.282, -79.927, -89.186, 4.347]
  MoveL 1357 to (445.86, -384.76, -5) mm, rotated rx -180 ry 0 rz -60 deg; joints [-19.353, -65.125, 150.557, -79.405, -88.959, 5.38]
  MoveC 1358 to (433.16, -397.46, -5) mm, rotated rx -180 ry 0 rz -60 deg; joints [-19.83, -64.661, 149.381, -79.893, -88.871, 6.087] to (420.46, -384.76, -5) mm, rotated rx 180 ry 0 rz -60 deg; joints [-18.84, -64.435, 148.816, -78.915, -88.717, 6.403]
  MoveL 1359 to (395.06, -384.76, -5) mm, rotated rx -180 ry 0 rz -30 deg; joints [-13.026, -67.809, 157.843, -43.031, -89.409, 0.647]
  MoveL 1360 to (318.86, -384.76, -5) mm, rotated rx 180 ry 0 rz -30 deg; joints [-11.92, -65.896, 152.536, -41.999, -86.884, 2.918]
  MoveC 1361 to (309.44, -397.03, -5) mm, rotated rx -180 ry 0 rz -5 deg; joints [-4.097, -67.286, 156.225, -9.105, -88.109, 0.515] to (293.46, -384.76, -5) mm, rotated rx -180 ry 0 rz 0 deg; joints [-1.268, -66.985, 155.328, -1.273, -87.473, 0.309]
  MoveL 1362 to (191.86, -384.76, -5) mm, rotated rx -180 ry 0 rz 0 deg; joints [-1.132, -64.166, 148.007, -1.144, -82.973, 0.395]
  MoveC 1363 to (179.16, -397.46, -5) mm, rotated rx -180 ry 0 rz 0 deg; joints [-1.87, -63.773, 147.055, -1.891, -82.416, 0.494] to (166.46, -384.76, -5) mm, rotated rx -180 ry 0 rz 0 deg; joints [-1.102, -63.406, 146.149, -1.118, -81.875, 0.414]
  MoveL 1364 to (90.26, -384.76, -5) mm, rotated rx -180 ry 0 rz 0 deg; joints [-1.022, -61.017, 140.499, -1.047, -78.614, 0.463]
  MoveL 1365 to (64.86, -384.76, -5) mm, rotated rx 180 ry 0 rz 0 deg; joints [-0.998, -60.188, 138.588, -1.026, -77.533, 0.479]
  MoveC 1366 to (61.14, -393.74, -5) mm, rotated rx -180 ry 0 rz 0 deg; joints [-1.47, -60.055, 138.292, -1.51, -77.371, 0.58] to (52.16, -397.46, -5) mm, rotated rx -180 ry 0 rz 0 deg; joints [-1.653, -59.753, 137.604, -1.7, -76.987, 0.63]
  MoveL 1367 to (52.16, -397.46, -5) mm, rotated rx -180 ry 0 rz 0 deg; joints [-1.653, -59.753, 137.604, -1.7, -76.987, 0.63]
  MoveC 1368 to (43.18, -393.74, -5) mm, rotated rx -180 ry 0 rz 0 deg; joints [-1.446, -59.457, 136.929, -1.49, -76.607, 0.596] to (39.46, -384.76, -5) mm, rotated rx -180 ry 0 rz 0 deg; joints [-0.975, -59.342, 136.661, -1.007, -76.451, 0.493]
  MoveL 1369 to (14.06, -384.76, -5) mm, rotated rx -180 ry 0 rz 0 deg; joints [-0.953, -58.481, 134.717, -0.989, -75.369, 0.508]
  MoveC 1370 to (13.61, -384.57, -5) mm, rotated rx 180 ry 0 rz 0 deg; joints [-0.943, -58.466, 134.683, -0.979, -75.35, 0.506] to (13.42, -384.12, -5) mm, rotated rx 180 ry 0 rz 0 deg; joints [-0.921, -58.46, 134.669, -0.956, -75.342, 0.5]
  MoveL 1371 to (13.42, -383.49, -5) mm, rotated rx 180 ry 0 rz 0 deg; joints [-0.888, -58.46, 134.67, -0.922, -75.342, 0.492]
  MoveC 1372 to (13.42, -383.04, -4.81) mm, rotated rx 180 ry 0 rz 0 deg; joints [-0.866, -58.475, 134.671, -0.899, -75.329, 0.487] to (13.42, -382.85, -4.37) mm, rotated rx 180 ry 0 rz 0 deg; joints [-0.856, -58.508, 134.672, -0.889, -75.296, 0.485]
  Set speed (500.0 mm/s)
  MoveL 1373 to (13.42, -382.85, 5) mm, rotated rx -180 ry 0 rz 0 deg; joints [-0.858, -59.203, 134.691, -0.895, -74.62, 0.497]
  MoveL 1374 to (12.15, -384.12, 5) mm, rotated rx -180 ry 0 rz 0 deg; joints [-0.922, -59.157, 134.592, -0.96, -74.567, 0.514]
  Set speed (25.4 mm/s)
  MoveL 1375 to (12.15, -384.12, 1) mm, rotated rx -180 ry 0 rz 0 deg; joints [-0.921, -58.862, 134.585, -0.958, -74.856, 0.509]
  MoveL 1376 to (12.15, -384.12, -7.71) mm, rotated rx 180 ry 0 rz 0 deg; joints [-0.919, -58.214, 134.564, -0.953, -75.482, 0.497]
  MoveC 1377 to (12.34, -384.12, -8.16) mm, rotated rx -180 ry 0 rz 0 deg; joints [-0.919, -58.187, 134.577, -0.953, -75.522, 0.497] to (12.79, -384.12, -8.35) mm, rotated rx -180 ry 0 rz 0 deg; joints [-0.919, -58.189, 134.611, -0.953, -75.555, 0.496]
  Set speed (50.8 mm/s)
  MoveL 1378 to (13.42, -384.12, -8.35) mm, rotated rx 180 ry 0 rz 0 deg; joints [-0.92, -58.21, 134.66, -0.954, -75.582, 0.496]
  MoveC 1379 to (13.87, -384.31, -8.35) mm, rotated rx 180 ry 0 rz 0 deg; joints [-0.93, -58.225, 134.695, -0.964, -75.602, 0.498] to (14.06, -384.76, -8.35) mm, rotated rx -180 ry 0 rz 0 deg; joints [-0.952, -58.231, 134.708, -0.987, -75.61, 0.503]
  MoveL 1380 to (14.06, -537.16, -8.35) mm, rotated rx -180 ry 0 rz 0 deg; joints [-8.614, -57.758, 133.725, -8.912, -75.259, 2.426]
  MoveL 1381 to (471.26, -537.16, -8.35) mm, rotated rx -180 ry 0 rz -60 deg; joints [-28.513, -63.708, 147.733, -88.545, -89.648, 6.862]
  MoveL 1382 to (471.26, -384.76, -8.35) mm, rotated rx -180 ry 0 rz -60 deg; joints [-19.893, -65.436, 152.27, -79.922, -89.246, 4.007]
  MoveL 1383 to (445.86, -384.76, -8.35) mm, rotated rx -180 ry 0 rz -60 deg; joints [-19.353, -64.783, 150.545, -79.399, -89.02, 5.055]
  MoveC 1384 to (433.16, -397.46, -8.35) mm, rotated rx -180 ry 0 rz -60 deg; joints [-19.83, -64.328, 149.37, -79.888, -88.928, 5.77] to (420.46, -384.76, -8.35) mm, rotated rx -180 ry 0 rz -60 deg; joints [-18.84, -64.106, 148.805, -78.908, -88.778, 6.091]
  MoveL 1385 to (395.06, -384.76, -8.35) mm, rotated rx -180 ry 0 rz -30 deg; joints [-13.026, -67.392, 157.829, -43.029, -89.703, 0.372]
  MoveL 1386 to (318.86, -384.76, -8.35) mm, rotated rx 180 ry 0 rz -30 deg; joints [-11.92, -65.536, 152.524, -41.986, -87.143, 2.685]
  MoveC 1387 to (309.44, -397.03, -8.35) mm, rotated rx -180 ry 0 rz -5 deg; joints [-4.096, -66.889, 156.211, -9.103, -88.488, 0.454] to (293.46, -384.76, -8.35) mm, rotated rx 180 ry 0 rz 0 deg; joints [-1.267, -66.598, 155.315, -1.271, -87.848, 0.301]
  MoveL 1388 to (191.86, -384.76, -8.35) mm, rotated rx 180 ry 0 rz 0 deg; joints [-1.131, -63.843, 147.996, -1.143, -83.284, 0.389]
  MoveC 1389 to (179.16, -397.46, -8.35) mm, rotated rx -180 ry 0 rz 0 deg; joints [-1.87, -63.457, 147.044, -1.889, -82.721, 0.483] to (166.46, -384.76, -8.35) mm, rotated rx -180 ry 0 rz 0 deg; joints [-1.102, -63.096, 146.138, -1.116, -82.174, 0.408]
  MoveL 1390 to (90.26, -384.76, -8.35) mm, rotated rx -180 ry 0 rz 0 deg; joints [-1.022, -60.741, 140.49, -1.045, -78.881, 0.458]
  MoveL 1391 to (64.86, -384.76, -8.35) mm, rotated rx 180 ry 0 rz 0 deg; joints [-0.997, -59.921, 138.578, -1.025, -77.79, 0.474]
  MoveC 1392 to (61.14, -393.74, -8.35) mm, rotated rx -180 ry 0 rz 0 deg; joints [-1.469, -59.79, 138.282, -1.508, -77.627, 0.573] to (52.16, -397.46, -8.35) mm, rotated rx -180 ry 0 rz 0 deg; joints [-1.652, -59.49, 137.595, -1.698, -77.24, 0.622]
  MoveL 1393 to (52.16, -397.46, -8.35) mm, rotated rx -180 ry 0 rz 0 deg; joints [-1.652, -59.49, 137.595, -1.698, -77.24, 0.622]
  MoveC 1394 to (43.18, -393.74, -8.35) mm, rotated rx -180 ry 0 rz 0 deg; joints [-1.445, -59.198, 136.92, -1.488, -76.857, 0.589] to (39.46, -384.76, -8.35) mm, rotated rx -180 ry 0 rz 0 deg; joints [-0.974, -59.084, 136.652, -1.005, -76.7, 0.489]
  MoveL 1395 to (14.06, -384.76, -8.35) mm, rotated rx -180 ry 0 rz 0 deg; joints [-0.952, -58.231, 134.708, -0.987, -75.61, 0.503]
  MoveC 1396 to (13.61, -384.57, -8.35) mm, rotated rx 180 ry 0 rz 0 deg; joints [-0.943, -58.216, 134.674, -0.977, -75.59, 0.501] to (13.42, -384.12, -8.35) mm, rotated rx 180 ry 0 rz 0 deg; joints [-0.92, -58.21, 134.66, -0.954, -75.582, 0.496]
  MoveL 1397 to (13.42, -383.49, -8.35) mm, rotated rx 180 ry 0 rz 0 deg; joints [-0.888, -58.211, 134.661, -0.921, -75.582, 0.488]
  MoveC 1398 to (13.42, -383.04, -8.16) mm, rotated rx -180 ry 0 rz 0 deg; joints [-0.865, -58.225, 134.662, -0.897, -75.569, 0.483] to (13.42, -382.85, -7.72) mm, rotated rx 180 ry 0 rz 0 deg; joints [-0.856, -58.259, 134.664, -0.888, -75.537, 0.481]
  Set speed (500.0 mm/s)
  MoveL 1399 to (13.42, -382.85, 6) mm, rotated rx -180 ry 0 rz 0 deg; joints [-0.859, -59.277, 134.692, -0.895, -74.547, 0.498]
  MoveL 1400 to (-13.42, -382.85, 6) mm, rotated rx -180 ry 0 rz 0 deg; joints [-0.839, -58.323, 132.618, -0.879, -73.427, 0.51]
  Set speed (25.4 mm/s)
  MoveL 1401 to (-13.42, -382.85, -4.37) mm, rotated rx -180 ry 0 rz 0 deg; joints [-0.836, -57.58, 132.599, -0.874, -74.151, 0.498]
  MoveC 1402 to (-13.42, -383.04, -4.81) mm, rotated rx -180 ry 0 rz 0 deg; joints [-0.845, -57.547, 132.598, -0.883, -74.183, 0.5] to (-13.42, -383.49, -5) mm, rotated rx 180 ry 0 rz 0 deg; joints [-0.868, -57.533, 132.597, -0.906, -74.195, 0.506]
  Set speed (50.8 mm/s)
  MoveL 1403 to (-13.42, -384.12, -5) mm, rotated rx -180 ry 0 rz 0 deg; joints [-0.899, -57.533, 132.596, -0.939, -74.195, 0.514]
  MoveC 1404 to (-13.61, -384.57, -5) mm, rotated rx -180 ry 0 rz 0 deg; joints [-0.921, -57.526, 132.581, -0.962, -74.187, 0.52] to (-14.06, -384.76, -5) mm, rotated rx -180 ry 0 rz 0 deg; joints [-0.93, -57.51, 132.546, -0.971, -74.168, 0.523]
  MoveL 1405 to (-39.46, -384.76, -5) mm, rotated rx -180 ry 0 rz 0 deg; joints [-0.91, -56.617, 130.564, -0.955, -73.08, 0.537]
  MoveC 1406 to (-52.16, -397.46, -5) mm, rotated rx -180 ry 0 rz 0 deg; joints [-1.508, -56.151, 129.545, -1.585, -72.53, 0.725] to (-64.86, -384.76, -5) mm, rotated rx -180 ry 0 rz 0 deg; joints [-0.891, -55.709, 128.563, -0.941, -71.987, 0.55]
  MoveL 1407 to (-90.26, -384.76, -5) mm, rotated rx -180 ry 0 rz 0 deg; joints [-0.872, -54.785, 126.54, -0.928, -70.888, 0.563]
  MoveL 1408 to (-166.46, -384.76, -5) mm, rotated rx -180 ry 0 rz 0 deg; joints [-0.821, -51.918, 120.333, -0.893, -67.548, 0.601]
  MoveC 1409 to (-179.16, -397.46, -5) mm, rotated rx -180 ry 0 rz 0 deg; joints [-1.363, -51.413, 119.256, -1.485, -66.98, 0.833] to (-191.86, -384.76, -5) mm, rotated rx 180 ry 0 rz 0 deg; joints [-0.806, -50.929, 118.212, -0.884, -66.416, 0.614]
  MoveL 1410 to (-293.46, -384.76, -5) mm, rotated rx -180 ry 0 rz 0 deg; joints [-0.748, -46.789, 109.419, -0.854, -61.763, 0.665]
  MoveC 1411 to (-306.16, -397.46, -5) mm, rotated rx -180 ry 0 rz 0 deg; joints [-1.243, -46.237, 108.26, -1.424, -61.161, 0.94] to (-318.86, -384.76, -5) mm, rotated rx 180 ry 0 rz 0 deg; joints [-0.735, -45.704, 107.132, -0.849, -60.561, 0.678]
  MoveL 1412 to (-395.06, -384.76, -5) mm, rotated rx -180 ry 0 rz 0 deg; joints [-0.699, -42.305, 100.01, -0.84, -56.838, 0.721]
  MoveL 1413 to (-420.46, -384.76, -5) mm, rotated rx 180 ry 0 rz 0 deg; joints [-0.687, -41.119, 97.537, -0.839, -55.551, 0.736]
  MoveC 1414 to (-433.16, -397.46, -5) mm, rotated rx 180 ry 0 rz 0 deg; joints [-1.143, -40.502, 96.259, -1.402, -54.895, 1.061] to (-445.86, -384.76, -5) mm, rotated rx -180 ry 0 rz 0 deg; joints [-0.676, -39.903, 95.006, -0.839, -54.237, 0.752]
  MoveL 1415 to (-471.26, -384.76, -5) mm, rotated rx 180 ry 0 rz 0 deg; joints [-0.666, -38.654, 92.414, -0.84, -52.893, 0.769]
  MoveL 1416 to (-471.26, -537.16, -5) mm, rotated rx -180 ry 0 rz 0 deg; joints [-6.048, -38.179, 91.483, -7.619, -52.675, 4.817]
  MoveL 1417 to (-14.06, -537.16, -5) mm, rotated rx -180 ry 0 rz 0 deg; joints [-8.408, -57.037, 131.576, -8.76, -73.841, 2.599]
  MoveL 1418 to (-14.06, -384.76, -5) mm, rotated rx -180 ry 0 rz 0 deg; joints [-0.93, -57.51, 132.546, -0.971, -74.168, 0.523]
  MoveC 1419 to (-13.87, -384.31, -5) mm, rotated rx 180 ry 0 rz 0 deg; joints [-0.908, -57.517, 132.561, -0.948, -74.176, 0.517] to (-13.42, -384.12, -5) mm, rotated rx -180 ry 0 rz 0 deg; joints [-0.899, -57.533, 132.596, -0.939, -74.195, 0.514]
  MoveL 1420 to (-12.79, -384.12, -5) mm, rotated rx -180 ry 0 rz 0 deg; joints [-0.9, -57.555, 132.645, -0.939, -74.223, 0.514]
  MoveC 1421 to (-12.34, -384.12, -4.81) mm, rotated rx -180 ry 0 rz 0 deg; joints [-0.9, -57.584, 132.68, -0.939, -74.229, 0.514] to (-12.15, -384.12, -4.37) mm, rotated rx -180 ry 0 rz 0 deg; joints [-0.9, -57.623, 132.696, -0.94, -74.205, 0.514]
  Set speed (500.0 mm/s)
  MoveL 1422 to (-12.15, -384.12, 5) mm, rotated rx 180 ry 0 rz 0 deg; joints [-0.902, -58.296, 132.714, -0.945, -73.551, 0.526]
  MoveL 1423 to (-13.42, -382.85, 5) mm, rotated rx -180 ry 0 rz 0 deg; joints [-0.838, -58.252, 132.617, -0.879, -73.497, 0.509]
  Set speed (25.4 mm/s)
  MoveL 1424 to (-13.42, -382.85, 1) mm, rotated rx -180 ry 0 rz 0 deg; joints [-0.838, -57.965, 132.61, -0.877, -73.777, 0.504]
  MoveL 1425 to (-13.42, -382.85, -7.72) mm, rotated rx -180 ry 0 rz 0 deg; joints [-0.836, -57.338, 132.59, -0.872, -74.384, 0.494]
  MoveC 1426 to (-13.42, -383.04, -8.16) mm, rotated rx -180 ry 0 rz 0 deg; joints [-0.845, -57.306, 132.589, -0.881, -74.415, 0.496] to (-13.42, -383.49, -8.35) mm, rotated rx -180 ry 0 rz 0 deg; joints [-0.867, -57.292, 132.588, -0.904, -74.428, 0.502]
  Set speed (50.8 mm/s)
  MoveL 1427 to (-13.42, -384.12, -8.35) mm, rotated rx 180 ry 0 rz 0 deg; joints [-0.898, -57.291, 132.587, -0.937, -74.428, 0.51]
  MoveC 1428 to (-13.61, -384.57, -8.35) mm, rotated rx 180 ry 0 rz 0 deg; joints [-0.92, -57.285, 132.572, -0.96, -74.42, 0.516] to (-14.06, -384.76, -8.35) mm, rotated rx -180 ry 0 rz 0 deg; joints [-0.929, -57.269, 132.537, -0.969, -74.401, 0.519]
  MoveL 1429 to (-39.46, -384.76, -8.35) mm, rotated rx 180 ry 0 rz 0 deg; joints [-0.909, -56.383, 130.556, -0.953, -73.305, 0.532]
  MoveC 1430 to (-52.16, -397.46, -8.35) mm, rotated rx -180 ry 0 rz 0 deg; joints [-1.508, -55.921, 129.536, -1.583, -72.752, 0.719] to (-64.86, -384.76, -8.35) mm, rotated rx -180 ry 0 rz 0 deg; joints [-0.89, -55.481, 128.554, -0.939, -72.206, 0.546]
  MoveL 1431 to (-90.26, -384.76, -8.35) mm, rotated rx 180 ry 0 rz 0 deg; joints [-0.872, -54.564, 126.532, -0.926, -71.101, 0.559]
  MoveL 1432 to (-166.46, -384.76, -8.35) mm, rotated rx 180 ry 0 rz 0 deg; joints [-0.821, -51.714, 120.325, -0.891, -67.744, 0.597]
  MoveC 1433 to (-179.16, -397.46, -8.35) mm, rotated rx -180 ry 0 rz 0 deg; joints [-1.363, -51.212, 119.248, -1.483, -67.173, 0.827] to (-191.86, -384.76, -8.35) mm, rotated rx 180 ry 0 rz 0 deg; joints [-0.805, -50.731, 118.204, -0.882, -66.606, 0.61]
  MoveL 1434 to (-293.46, -384.76, -8.35) mm, rotated rx -180 ry 0 rz 0 deg; joints [-0.748, -46.609, 109.411, -0.852, -61.935, 0.662]
  MoveC 1435 to (-306.16, -397.46, -8.35) mm, rotated rx 180 ry 0 rz 0 deg; joints [-1.243, -46.059, 108.253, -1.421, -61.331, 0.935] to (-318.86, -384.76, -8.35) mm, rotated rx -180 ry 0 rz 0 deg; joints [-0.735, -45.528, 107.124, -0.847, -60.729, 0.675]
  MoveL 1436 to (-395.06, -384.76, -8.35) mm, rotated rx -180 ry 0 rz 0 deg; joints [-0.698, -42.14, 100.002, -0.837, -56.996, 0.718]
  MoveL 1437 to (-420.46, -384.76, -8.35) mm, rotated rx -180 ry 0 rz 0 deg; joints [-0.687, -40.957, 97.529, -0.836, -55.705, 0.733]
  MoveC 1438 to (-433.16, -397.46, -8.35) mm, rotated rx -180 ry 0 rz 0 deg; joints [-1.143, -40.342, 96.251, -1.399, -55.047, 1.056] to (-445.86, -384.76, -8.35) mm, rotated rx 180 ry 0 rz 0 deg; joints [-0.676, -39.744, 94.999, -0.836, -54.388, 0.749]
  MoveL 1439 to (-471.26, -384.76, -8.35) mm, rotated rx -180 ry 0 rz 0 deg; joints [-0.665, -38.499, 92.406, -0.837, -53.041, 0.766]
  MoveL 1440 to (-471.26, -537.16, -8.35) mm, rotated rx -180 ry 0 rz 0 deg; joints [-6.048, -38.025, 91.476, -7.603, -52.821, 4.792]
  MoveL 1441 to (-14.06, -537.16, -8.35) mm, rotated rx 180 ry 0 rz 0 deg; joints [-8.408, -56.799, 131.567, -8.749, -74.067, 2.563]
  MoveL 1442 to (-14.06, -384.76, -8.35) mm, rotated rx 180 ry 0 rz 0 deg; joints [-0.929, -57.269, 132.537, -0.969, -74.401, 0.519]
  MoveC 1443 to (-13.87, -384.31, -8.35) mm, rotated rx -180 ry 0 rz 0 deg; joints [-0.907, -57.276, 132.552, -0.946, -74.409, 0.513] to (-13.42, -384.12, -8.35) mm, rotated rx 180 ry 0 rz 0 deg; joints [-0.898, -57.291, 132.587, -0.937, -74.428, 0.51]
  MoveL 1444 to (-12.79, -384.12, -8.35) mm, rotated rx 180 ry 0 rz 0 deg; joints [-0.899, -57.313, 132.636, -0.937, -74.455, 0.51]
  MoveC 1445 to (-12.34, -384.12, -8.16) mm, rotated rx -180 ry 0 rz 0 deg; joints [-0.899, -57.342, 132.672, -0.938, -74.462, 0.51] to (-12.15, -384.12, -7.72) mm, rotated rx 180 ry 0 rz 0 deg; joints [-0.899, -57.381, 132.687, -0.938, -74.439, 0.51]
  Set speed (500.0 mm/s)
  MoveL 1446 to (-12.15, -384.12, 6) mm, rotated rx -180 ry 0 rz 0 deg; joints [-0.903, -58.368, 132.716, -0.946, -73.48, 0.527]
  MoveL 1447 to (-52.79, 196.51, 6) mm, rotated rx -180 ry 0 rz 0 deg; joints [25.164, -52.399, 119.385, 27.203, -68.421, -10.024]
  Set speed (25.4 mm/s)
  MoveL 1448 to (-52.79, 196.51, -4.37) mm, rotated rx -180 ry 0 rz 0 deg; joints [25.169, -51.781, 119.369, 27.101, -68.957, -9.731]
  MoveC 1449 to (-52.79, 196.7, -4.81) mm, rotated rx 180 ry 0 rz 0 deg; joints [25.176, -51.751, 119.362, 27.105, -68.978, -9.723] to (-52.79, 197.15, -5) mm, rotated rx 180 ry 0 rz 0 deg; joints [25.194, -51.733, 119.345, 27.123, -68.983, -9.728]
  Set speed (50.8 mm/s)
  MoveL 1450 to (-52.79, 197.78, -5) mm, rotated rx -180 ry 0 rz 0 deg; joints [25.219, -51.723, 119.323, 27.151, -68.976, -9.743]
  MoveC 1451 to (-52.61, 198.23, -5) mm, rotated rx -180 ry 0 rz 0 deg; joints [25.24, -51.722, 119.321, 27.174, -68.979, -9.752] to (-52.16, 198.42, -5) mm, rotated rx 180 ry 0 rz 0 deg; joints [25.256, -51.735, 119.348, 27.188, -68.994, -9.75]
  MoveL 1452 to (-14.06, 198.42, -5) mm, rotated rx -180 ry 0 rz 0 deg; joints [25.978, -53.07, 122.192, 27.69, -70.456, -9.261]
  MoveL 1453 to (-14.06, 350.82, -5) mm, rotated rx 180 ry 0 rz 0 deg; joints [31.751, -50.283, 116.037, 34.376, -68.715, -13.136]
  MoveL 1454 to (-39.46, 350.82, -5) mm, rotated rx -180 ry 0 rz 0 deg; joints [31.198, -49.399, 114.178, 34.016, -67.778, -13.52]
  MoveC 1455 to (-52.16, 338.12, -5) mm, rotated rx -180 ry 0 rz 0 deg; joints [30.478, -49.208, 113.798, 33.303, -67.45, -13.356] to (-64.86, 350.82, -5) mm, rotated rx -180 ry 0 rz 0 deg; joints [30.661, -48.496, 112.285, 33.682, -66.826, -13.908]
  MoveL 1456 to (-90.26, 350.82, -5) mm, rotated rx -180 ry 0 rz 0 deg; joints [30.142, -47.574, 110.355, 33.377, -65.857, -14.303]
  MoveL 1457 to (-166.46, 350.82, -5) mm, rotated rx 180 ry 0 rz 0 deg; joints [28.674, -44.685, 104.332, 32.625, -62.844, -15.539]
  MoveC 1458 to (-179.16, 338.12, -5) mm, rotated rx 180 ry 0 rz 0 deg; joints [28.015, -44.446, 103.852, 31.978, -62.462, -15.366] to (-191.86, 350.82, -5) mm, rotated rx -180 ry 0 rz 0 deg; joints [28.214, -43.678, 102.239, 32.432, -61.802, -15.973]
  MoveL 1459 to (-293.46, 350.82, -5) mm, rotated rx -180 ry 0 rz 0 deg; joints [26.501, -39.391, 93.371, 31.966, -57.417, -17.869]
  MoveC 1460 to (-306.16, 338.12, -5) mm, rotated rx -180 ry 0 rz 0 deg; joints [25.895, -39.096, 92.776, 31.383, -56.975, -17.695] to (-318.86, 350.82, -5) mm, rotated rx -180 ry 0 rz 0 deg; joints [26.102, -38.247, 91.011, 31.934, -56.26, -18.397]
  MoveL 1461 to (-395.06, 350.82, -5) mm, rotated rx 180 ry 0 rz 0 deg; joints [24.971, -34.597, 83.506, 32.085, -52.612, -20.164]
  MoveL 1462 to (-420.46, 350.82, -5) mm, rotated rx -180 ry 0 rz 0 deg; joints [24.614, -33.297, 80.839, 32.231, -51.328, -20.832]
  MoveC 1463 to (-433.16, 338.12, -5) mm, rotated rx 180 ry 0 rz 0 deg; joints [24.056, -32.926, 80.09, 31.722, -50.808, -20.677] to (-445.86, 350.82, -5) mm, rotated rx -180 ry 0 rz 0 deg; joints [24.267, -31.947, 78.073, 32.433, -50.005, -21.551]
  MoveL 1464 to (-471.26, 350.82, -5) mm, rotated rx -180 ry 0 rz 0 deg; joints [23.928, -30.542, 75.197, 32.701, -48.637, -22.331]
  MoveL 1465 to (-471.26, 198.42, -5) mm, rotated rx 180 ry 0 rz 0 deg; joints [19.259, -33.784, 81.98, 25.428, -50.169, -16.361]
  MoveL 1466 to (-445.86, 198.42, -5) mm, rotated rx -180 ry 0 rz 0 deg; joints [19.543, -35.113, 84.713, 25.29, -51.517, -15.804]
  MoveL 1467 to (-52.16, 198.42, -5) mm, rotated rx 180 ry 0 rz 0 deg; joints [25.256, -51.735, 119.348, 27.188, -68.994, -9.75]
  MoveC 1468 to (-51.71, 198.23, -5) mm, rotated rx 180 ry 0 rz 0 deg; joints [25.257, -51.754, 119.389, 27.185, -69.014, -9.74] to (-51.52, 197.78, -5) mm, rotated rx -180 ry 0 rz 0 deg; joints [25.242, -51.768, 119.419, 27.167, -69.026, -9.727]
  MoveL 1469 to (-51.52, 197.15, -5) mm, rotated rx -180 ry 0 rz 0 deg; joints [25.218, -51.778, 119.441, 27.139, -69.032, -9.712]
  MoveC 1470 to (-51.52, 196.7, -4.81) mm, rotated rx 180 ry 0 rz 0 deg; joints [25.2, -51.796, 119.457, 27.12, -69.028, -9.707] to (-51.52, 196.52, -4.37) mm, rotated rx -180 ry 0 rz 0 deg; joints [25.192, -51.826, 119.465, 27.116, -69.006, -9.715]
  Set speed (500.0 mm/s)
  MoveL 1471 to (-51.52, 196.51, 5) mm, rotated rx -180 ry 0 rz 0 deg; joints [25.188, -52.385, 119.48, 27.208, -68.521, -9.98]
  MoveL 1472 to (-52.79, 196.51, 5) mm, rotated rx -180 ry 0 rz 0 deg; joints [25.165, -52.34, 119.384, 27.193, -68.473, -9.996]
  Set speed (25.4 mm/s)
  MoveL 1473 to (-52.79, 196.52, 1) mm, rotated rx -180 ry 0 rz 0 deg; joints [25.166, -52.101, 119.379, 27.153, -68.68, -9.882]
  MoveL 1474 to (-52.79, 196.52, -7.71) mm, rotated rx -180 ry 0 rz 0 deg; joints [25.17, -51.58, 119.362, 27.068, -69.13, -9.637]
  MoveC 1475 to (-52.79, 196.7, -8.16) mm, rotated rx -180 ry 0 rz 0 deg; joints [25.178, -51.55, 119.354, 27.073, -69.151, -9.629] to (-52.79, 197.15, -8.35) mm, rotated rx -180 ry 0 rz 0 deg; joints [25.196, -51.532, 119.338, 27.091, -69.155, -9.635]
  Set speed (50.8 mm/s)
  MoveL 1476 to (-52.79, 197.78, -8.35) mm, rotated rx 180 ry 0 rz 0 deg; joints [25.221, -51.522, 119.315, 27.119, -69.149, -9.65]
  MoveC 1477 to (-52.61, 198.23, -8.35) mm, rotated rx -180 ry 0 rz 0 deg; joints [25.242, -51.521, 119.313, 27.142, -69.151, -9.658] to (-52.16, 198.42, -8.35) mm, rotated rx -180 ry 0 rz 0 deg; joints [25.257, -51.534, 119.341, 27.156, -69.167, -9.656]
  MoveL 1478 to (-14.06, 198.42, -8.35) mm, rotated rx 180 ry 0 rz 0 deg; joints [25.98, -52.862, 122.184, 27.659, -70.634, -9.163]
  MoveL 1479 to (-14.06, 350.82, -8.35) mm, rotated rx -180 ry 0 rz 0 deg; joints [31.753, -50.09, 116.03, 34.337, -68.868, -13.024]
  MoveL 1480 to (-39.46, 350.82, -8.35) mm, rotated rx -180 ry 0 rz 0 deg; joints [31.199, -49.21, 114.171, 33.976, -67.93, -13.411]
  MoveC 1481 to (-52.16, 338.12, -8.35) mm, rotated rx -180 ry 0 rz 0 deg; joints [30.479, -49.02, 113.791, 33.263, -67.602, -13.249] to (-64.86, 350.82, -8.35) mm, rotated rx 180 ry 0 rz 0 deg; joints [30.663, -48.311, 112.278, 33.642, -66.975, -13.802]
  MoveL 1482 to (-90.26, 350.82, -8.35) mm, rotated rx 180 ry 0 rz 0 deg; joints [30.143, -47.393, 110.348, 33.335, -66.003, -14.199]
  MoveL 1483 to (-166.46, 350.82, -8.35) mm, rotated rx -180 ry 0 rz 0 deg; joints [28.676, -44.514, 104.325, 32.582, -62.983, -15.441]
  MoveC 1484 to (-179.16, 338.12, -8.35) mm, rotated rx -180 ry 0 rz 0 deg; joints [28.017, -44.276, 103.845, 31.934, -62.601, -15.269] to (-191.86, 350.82, -8.35) mm, rotated rx -180 ry 0 rz 0 deg; joints [28.215, -43.51, 102.232, 32.387, -61.938, -15.876]
  MoveL 1485 to (-293.46, 350.82, -8.35) mm, rotated rx -180 ry 0 rz 0 deg; joints [26.502, -39.235, 93.364, 31.917, -57.544, -17.777]
  MoveC 1486 to (-306.16, 338.12, -8.35) mm, rotated rx -180 ry 0 rz 0 deg; joints [25.897, -38.94, 92.769, 31.334, -57.102, -17.604] to (-318.86, 350.82, -8.35) mm, rotated rx -180 ry 0 rz 0 deg; joints [26.103, -38.093, 91.004, 31.884, -56.385, -18.305]
  MoveL 1487 to (-395.06, 350.82, -8.35) mm, rotated rx 180 ry 0 rz 0 deg; joints [24.972, -34.451, 83.499, 32.031, -52.73, -20.072]
  MoveL 1488 to (-420.46, 350.82, -8.35) mm, rotated rx 180 ry 0 rz 0 deg; joints [24.615, -33.153, 80.831, 32.174, -51.444, -20.74]
  MoveC 1489 to (-433.16, 338.12, -8.35) mm, rotated rx -180 ry 0 rz 0 deg; joints [24.057, -32.783, 80.082, 31.666, -50.923, -20.586] to (-445.86, 350.82, -8.35) mm, rotated rx 180 ry 0 rz 0 deg; joints [24.268, -31.806, 78.066, 32.375, -50.118, -21.459]
  MoveL 1490 to (-471.26, 350.82, -8.35) mm, rotated rx 180 ry 0 rz 0 deg; joints [23.93, -30.403, 75.189, 32.64, -48.748, -22.238]
  MoveL 1491 to (-471.26, 198.42, -8.35) mm, rotated rx -180 ry 0 rz 0 deg; joints [19.26, -33.639, 81.973, 25.38, -50.293, -16.285]
  MoveL 1492 to (-445.86, 198.42, -8.35) mm, rotated rx 180 ry 0 rz 0 deg; joints [19.544, -34.966, 84.706, 25.245, -51.643, -15.729]
  MoveL 1493 to (-52.16, 198.42, -8.35) mm, rotated rx 180 ry 0 rz 0 deg; joints [25.257, -51.534, 119.341, 27.156, -69.167, -9.656]
  MoveC 1494 to (-51.71, 198.23, -8.35) mm, rotated rx 180 ry 0 rz 0 deg; joints [25.258, -51.553, 119.381, 27.153, -69.186, -9.646] to (-51.52, 197.78, -8.35) mm, rotated rx -180 ry 0 rz 0 deg; joints [25.244, -51.567, 119.411, 27.135, -69.198, -9.633]
  MoveL 1495 to (-51.52, 197.15, -8.35) mm, rotated rx -180 ry 0 rz 0 deg; joints [25.219, -51.577, 119.434, 27.107, -69.205, -9.618]
  MoveC 1496 to (-51.52, 196.7, -8.16) mm, rotated rx -180 ry 0 rz 0 deg; joints [25.201, -51.595, 119.45, 27.088, -69.2, -9.613] to (-51.52, 196.52, -7.72) mm, rotated rx 180 ry 0 rz 0 deg; joints [25.194, -51.625, 119.458, 27.084, -69.179, -9.621]
  Set speed (500.0 mm/s)
  MoveL 1497 to (-51.52, 196.51, 6) mm, rotated rx -180 ry 0 rz 0 deg; joints [25.187, -52.445, 119.481, 27.218, -68.47, -10.008]
  MoveL 1498 to (18.41, 196.51, 6) mm, rotated rx -180 ry 0 rz 0 deg; joints [26.542, -54.911, 124.651, 28.178, -71.095, -9.14]
  Set speed (25.4 mm/s)
  MoveL 1499 to (18.41, 196.51, -4.36) mm, rotated rx -180 ry 0 rz 0 deg; joints [26.547, -54.25, 124.634, 28.081, -71.664, -8.821]
  MoveC 1500 to (18.41, 196.7, -4.81) mm, rotated rx -180 ry 0 rz 0 deg; joints [26.555, -54.218, 124.627, 28.085, -71.687, -8.812] to (18.41, 197.15, -5) mm, rotated rx 180 ry 0 rz 0 deg; joints [26.573, -54.199, 124.61, 28.104, -71.692, -8.816]
  Set speed (50.8 mm/s)
  MoveL 1501 to (18.41, 197.78, -5) mm, rotated rx -180 ry 0 rz 0 deg; joints [26.599, -54.189, 124.587, 28.133, -71.684, -8.83]
  MoveC 1502 to (18.6, 198.23, -5) mm, rotated rx 180 ry 0 rz 0 deg; joints [26.621, -54.188, 124.584, 28.156, -71.686, -8.838] to (19.05, 198.42, -5) mm, rotated rx -180 ry 0 rz 0 deg; joints [26.638, -54.2, 124.61, 28.171, -71.701, -8.837]
  MoveL 1503 to (39.46, 198.42, -5) mm, rotated rx -180 ry 0 rz 0 deg; joints [27.061, -54.883, 126.078, 28.49, -72.458, -8.574]
  MoveL 1504 to (471.26, 198.42, -5) mm, rotated rx -180 ry 0 rz 0 deg; joints [39.981, -66.913, 153.4, 40.065, -86.439, -1.989]
  MoveL 1505 to (471.26, 350.82, -5) mm, rotated rx 180 ry 0 rz 0 deg; joints [46.803, -64.001, 145.794, 47.184, -83.527, -5.739]
  MoveL 1506 to (445.86, 350.82, -5) mm, rotated rx -180 ry 0 rz 0 deg; joints [45.743, -63.431, 144.5, 46.186, -82.916, -6.16]
  MoveC 1507 to (433.16, 338.12, -5) mm, rotated rx -180 ry 0 rz 0 deg; joints [44.715, -63.411, 144.504, 45.154, -82.819, -6.03] to (420.46, 350.82, -5) mm, rotated rx 180 ry 0 rz 0 deg; joints [44.72, -62.844, 143.175, 45.23, -82.282, -6.577]
  MoveL 1508 to (395.06, 350.82, -5) mm, rotated rx 180 ry 0 rz 0 deg; joints [43.732, -62.24, 141.82, 44.315, -81.628, -6.987]
  MoveL 1509 to (318.86, 350.82, -5) mm, rotated rx 180 ry 0 rz 0 deg; joints [40.971, -60.329, 137.58, 41.805, -79.548, -8.188]
  MoveC 1510 to (306.16, 338.12, -5) mm, rotated rx 180 ry 0 rz 0 deg; joints [40.033, -60.263, 137.473, 40.867, -79.38, -8.057] to (293.46, 350.82, -5) mm, rotated rx -180 ry 0 rz 0 deg; joints [40.113, -59.66, 136.11, 41.044, -78.818, -8.578]
  MoveL 1511 to (191.86, 350.82, -5) mm, rotated rx -180 ry 0 rz 0 deg; joints [36.965, -56.823, 129.947, 38.341, -75.733, -10.103]
  MoveC 1512 to (179.16, 338.12, -5) mm, rotated rx -180 ry 0 rz 0 deg; joints [36.113, -56.712, 129.739, 37.49, -75.503, -9.963] to (166.46, 350.82, -5) mm, rotated rx -180 ry 0 rz 0 deg; joints [36.244, -56.074, 128.336, 37.747, -74.921, -10.478]
  MoveL 1513 to (90.26, 350.82, -5) mm, rotated rx 180 ry 0 rz 0 deg; joints [34.219, -53.732, 123.331, 36.147, -72.395, -11.594]
  MoveL 1514 to (64.86, 350.82, -5) mm, rotated rx -180 ry 0 rz 0 deg; joints [33.587, -52.918, 121.603, 35.672, -71.523, -11.967]
  MoveC 1515 to (61.14, 341.84, -5) mm, rotated rx 180 ry 0 rz 0 deg; joints [33.165, -52.981, 121.754, 35.219, -71.505, -11.782] to (52.16, 338.12, -5) mm, rotated rx -180 ry 0 rz 0 deg; joints [32.811, -52.764, 121.3, 34.9, -71.238, -11.814]
  MoveL 1516 to (52.16, 338.12, -5) mm, rotated rx -180 ry 0 rz 0 deg; joints [32.811, -52.764, 121.3, 34.9, -71.238, -11.814]
  MoveC 1517 to (43.18, 341.84, -5) mm, rotated rx 180 ry 0 rz 0 deg; joints [32.735, -52.394, 120.509, 34.904, -70.876, -12.044] to (39.46, 350.82, -5) mm, rotated rx -180 ry 0 rz 0 deg; joints [32.976, -52.088, 119.845, 35.225, -70.635, -12.341]
  MoveL 1518 to (14.06, 350.82, -5) mm, rotated rx -180 ry 0 rz 0 deg; joints [32.384, -51.241, 118.056, 34.807, -69.732, -12.717]
  MoveL 1519 to (14.06, 198.42, -5) mm, rotated rx 180 ry 0 rz 0 deg; joints [26.537, -54.032, 124.248, 28.096, -71.515, -8.901]
  MoveL 1520 to (19.04, 198.42, -5) mm, rotated rx -180 ry 0 rz 0 deg; joints [26.638, -54.2, 124.61, 28.171, -71.701, -8.837]
  MoveC 1521 to (19.49, 198.23, -5) mm, rotated rx -180 ry 0 rz 0 deg; joints [26.64, -54.218, 124.649, 28.17, -71.72, -8.827] to (19.68, 197.78, -5) mm, rotated rx -180 ry 0 rz 0 deg; joints [26.625, -54.232, 124.679, 28.152, -71.732, -8.814]
  MoveL 1522 to (19.68, 197.15, -5) mm, rotated rx -180 ry 0 rz 0 deg; joints [26.599, -54.242, 124.702, 28.123, -71.739, -8.8]
  MoveC 1523 to (19.68, 196.7, -4.81) mm, rotated rx 180 ry 0 rz 0 deg; joints [26.581, -54.261, 124.718, 28.105, -71.734, -8.795] to (19.68, 196.52, -4.37) mm, rotated rx -180 ry 0 rz 0 deg; joints [26.573, -54.293, 124.726, 28.1, -71.711, -8.805]
  Set speed (500.0 mm/s)
  MoveL 1524 to (19.68, 196.51, 5) mm, rotated rx 180 ry 0 rz 0 deg; joints [26.568, -54.891, 124.742, 28.188, -71.197, -9.093]
  MoveL 1525 to (18.41, 196.52, 5) mm, rotated rx -180 ry 0 rz 0 deg; joints [26.543, -54.848, 124.65, 28.168, -71.15, -9.109]
  Set speed (25.4 mm/s)
  MoveL 1526 to (18.41, 196.51, 1) mm, rotated rx -180 ry 0 rz 0 deg; joints [26.545, -54.593, 124.644, 28.131, -71.37, -8.986]
  MoveL 1527 to (18.41, 196.52, -7.72) mm, rotated rx -180 ry 0 rz 0 deg; joints [26.549, -54.035, 124.627, 28.051, -71.847, -8.719]
  MoveC 1528 to (18.41, 196.7, -8.16) mm, rotated rx 180 ry 0 rz 0 deg; joints [26.557, -54.004, 124.619, 28.055, -71.87, -8.709] to (18.41, 197.15, -8.35) mm, rotated rx -180 ry 0 rz 0 deg; joints [26.575, -53.984, 124.602, 28.074, -71.875, -8.714]
  Set speed (50.8 mm/s)
  MoveL 1529 to (18.41, 197.78, -8.35) mm, rotated rx -180 ry 0 rz 0 deg; joints [26.601, -53.974, 124.579, 28.103, -71.867, -8.728]
  MoveC 1530 to (18.6, 198.23, -8.35) mm, rotated rx -180 ry 0 rz 0 deg; joints [26.623, -53.973, 124.576, 28.126, -71.869, -8.736] to (19.05, 198.42, -8.35) mm, rotated rx -180 ry 0 rz 0 deg; joints [26.64, -53.985, 124.602, 28.141, -71.884, -8.734]
  MoveL 1531 to (39.46, 198.42, -8.35) mm, rotated rx 180 ry 0 rz 0 deg; joints [27.062, -54.664, 126.07, 28.46, -72.644, -8.469]
  MoveL 1532 to (471.26, 198.42, -8.35) mm, rotated rx -180 ry 0 rz 0 deg; joints [39.984, -66.546, 153.388, 40.054, -86.712, -1.759]
  MoveL 1533 to (471.26, 350.82, -8.35) mm, rotated rx -180 ry 0 rz 0 deg; joints [46.806, -63.694, 145.785, 47.163, -83.73, -5.519]
  MoveL 1534 to (445.86, 350.82, -8.35) mm, rotated rx -180 ry 0 rz 0 deg; joints [45.746, -63.132, 144.491, 46.163, -83.116, -5.95]
  MoveC 1535 to (433.16, 338.12, -8.35) mm, rotated rx -180 ry 0 rz 0 deg; joints [44.717, -63.112, 144.495, 45.131, -83.024, -5.824] to (420.46, 350.82, -8.35) mm, rotated rx 180 ry 0 rz 0 deg; joints [44.722, -62.553, 143.166, 45.206, -82.481, -6.375]
  MoveL 1536 to (395.06, 350.82, -8.35) mm, rotated rx 180 ry 0 rz 0 deg; joints [43.735, -61.957, 141.811, 44.29, -81.824, -6.794]
  MoveL 1537 to (318.86, 350.82, -8.35) mm, rotated rx 180 ry 0 rz 0 deg; joints [40.973, -60.067, 137.572, 41.777, -79.737, -8.016]
  MoveC 1538 to (306.16, 338.12, -8.35) mm, rotated rx -180 ry 0 rz 0 deg; joints [40.035, -60.001, 137.464, 40.839, -79.572, -7.889] to (293.46, 350.82, -8.35) mm, rotated rx -180 ry 0 rz 0 deg; joints [40.115, -59.404, 136.102, 41.014, -79.005, -8.413]
  MoveL 1539 to (191.86, 350.82, -8.35) mm, rotated rx -180 ry 0 rz 0 deg; joints [36.968, -56.591, 129.94, 38.308, -75.908, -9.961]
  MoveC 1540 to (179.16, 338.12, -8.35) mm, rotated rx -180 ry 0 rz 0 deg; joints [36.115, -56.481, 129.731, 37.457, -75.68, -9.824] to (166.46, 350.82, -8.35) mm, rotated rx 180 ry 0 rz 0 deg; joints [36.246, -55.848, 128.329, 37.713, -75.094, -10.34]
  MoveL 1541 to (90.26, 350.82, -8.35) mm, rotated rx 180 ry 0 rz 0 deg; joints [34.22, -53.521, 123.323, 36.111, -72.56, -11.469]
  MoveL 1542 to (64.86, 350.82, -8.35) mm, rotated rx -180 ry 0 rz 0 deg; joints [33.589, -52.712, 121.596, 35.635, -71.685, -11.845]
  MoveC 1543 to (61.14, 341.84, -8.35) mm, rotated rx -180 ry 0 rz 0 deg; joints [33.167, -52.774, 121.746, 35.183, -71.669, -11.661] to (52.16, 338.12, -8.35) mm, rotated rx -180 ry 0 rz 0 deg; joints [32.813, -52.558, 121.292, 34.864, -71.401, -11.695]
  MoveL 1544 to (52.16, 338.12, -8.35) mm, rotated rx 180 ry 0 rz 0 deg; joints [32.813, -52.558, 121.292, 34.864, -71.401, -11.695]
  MoveC 1545 to (43.18, 341.84, -8.35) mm, rotated rx -180 ry 0 rz 0 deg; joints [32.736, -52.191, 120.502, 34.867, -71.038, -11.926] to (39.46, 350.82, -8.35) mm, rotated rx 180 ry 0 rz 0 deg; joints [32.978, -51.886, 119.838, 35.188, -70.795, -12.222]
  MoveL 1546 to (14.06, 350.82, -8.35) mm, rotated rx -180 ry 0 rz 0 deg; joints [32.386, -51.044, 118.048, 34.769, -69.889, -12.601]
  MoveL 1547 to (14.06, 198.42, -8.35) mm, rotated rx 180 ry 0 rz 0 deg; joints [26.538, -53.818, 124.241, 28.066, -71.697, -8.799]
  MoveL 1548 to (19.05, 198.42, -8.35) mm, rotated rx -180 ry 0 rz 0 deg; joints [26.64, -53.985, 124.602, 28.141, -71.884, -8.734]
  MoveC 1549 to (19.49, 198.23, -8.35) mm, rotated rx 180 ry 0 rz 0 deg; joints [26.641, -54.003, 124.641, 28.139, -71.903, -8.724] to (19.68, 197.78, -8.35) mm, rotated rx 180 ry 0 rz 0 deg; joints [26.627, -54.017, 124.671, 28.122, -71.915, -8.712]
  MoveL 1550 to (19.68, 197.15, -8.35) mm, rotated rx -180 ry 0 rz 0 deg; joints [26.601, -54.027, 124.694, 28.093, -71.922, -8.697]
  MoveC 1551 to (19.68, 196.7, -8.16) mm, rotated rx 180 ry 0 rz 0 deg; joints [26.583, -54.046, 124.711, 28.074, -71.917, -8.693] to (19.68, 196.52, -7.72) mm, rotated rx -180 ry 0 rz 0 deg; joints [26.575, -54.078, 124.719, 28.07, -71.895, -8.703]
  Set speed (500.0 mm/s)
  MoveL 1552 to (19.68, 196.52, 6) mm, rotated rx 180 ry 0 rz 0 deg; joints [26.568, -54.955, 124.743, 28.197, -71.142, -9.124]
  MoveL 1553 to (18.41, 382.85, 6) mm, rotated rx -180 ry 0 rz 0 deg; joints [33.624, -51.352, 116.908, 36.37, -69, -13.934]
  Set speed (25.4 mm/s)
  MoveL 1554 to (18.41, 382.85, -4.37) mm, rotated rx -180 ry 0 rz 0 deg; joints [33.629, -50.752, 116.892, 36.244, -69.472, -13.566]
  MoveC 1555 to (18.41, 383.04, -4.81) mm, rotated rx 180 ry 0 rz 0 deg; joints [33.636, -50.722, 116.882, 36.247, -69.49, -13.556] to (18.41, 383.49, -5) mm, rotated rx -180 ry 0 rz 0 deg; joints [33.652, -50.702, 116.861, 36.264, -69.493, -13.562]
  Set speed (50.8 mm/s)
  MoveL 1556 to (18.41, 384.12, -5) mm, rotated rx -180 ry 0 rz 0 deg; joints [33.674, -50.688, 116.831, 36.291, -69.485, -13.58]
  MoveC 1557 to (18.6, 384.57, -5) mm, rotated rx -180 ry 0 rz 0 deg; joints [33.694, -50.685, 116.823, 36.312, -69.487, -13.59] to (19.05, 384.76, -5) mm, rotated rx -180 ry 0 rz 0 deg; joints [33.711, -50.696, 116.846, 36.328, -69.5, -13.588]
  MoveL 1558 to (64.86, 384.76, -5) mm, rotated rx -180 ry 0 rz 0 deg; joints [34.819, -52.204, 120.026, 37.114, -71.099, -12.895]
  MoveL 1559 to (471.26, 384.76, -5) mm, rotated rx -180 ry 0 rz 0 deg; joints [48.123, -63.25, 143.951, 48.602, -82.944, -6.69]
  MoveL 1560 to (471.26, 537.16, -5) mm, rotated rx -180 ry 0 rz 0 deg; joints [53.306, -59.465, 135.063, 54.352, -80.6, -11.39]
  MoveL 1561 to (445.86, 537.16, -5) mm, rotated rx -180 ry 0 rz 0 deg; joints [52.284, -58.911, 133.88, 53.424, -80.02, -11.75]
  MoveC 1562 to (433.16, 524.46, -5) mm, rotated rx -180 ry 0 rz 0 deg; joints [51.388, -58.966, 134.044, 52.518, -79.901, -11.52] to (420.46, 537.16, -5) mm, rotated rx -180 ry 0 rz 0 deg; joints [51.289, -58.34, 132.663, 52.529, -79.42, -12.113]
  MoveL 1563 to (395.06, 537.16, -5) mm, rotated rx -180 ry 0 rz 0 deg; joints [50.321, -57.753, 131.413, 51.668, -78.803, -12.479]
  MoveL 1564 to (318.86, 537.16, -5) mm, rotated rx -180 ry 0 rz 0 deg; joints [47.574, -55.89, 127.462, 49.281, -76.842, -13.591]
  MoveC 1565 to (306.16, 524.46, -5) mm, rotated rx -180 ry 0 rz 0 deg; joints [46.734, -55.897, 127.516, 48.434, -76.672, -13.376] to (293.46, 537.16, -5) mm, rotated rx -180 ry 0 rz 0 deg; joints [46.709, -55.236, 126.08, 48.549, -76.153, -13.967]
  MoveL 1566 to (191.86, 537.16, -5) mm, rotated rx 180 ry 0 rz 0 deg; joints [43.479, -52.452, 120.222, 45.933, -73.228, -15.503]
  MoveC 1567 to (179.16, 524.46, -5) mm, rotated rx -180 ry 0 rz 0 deg; joints [42.696, -52.414, 120.171, 45.147, -73.008, -15.295] to (166.46, 537.16, -5) mm, rotated rx -180 ry 0 rz 0 deg; joints [42.727, -51.713, 118.674, 45.354, -72.456, -15.897]
  MoveL 1568 to (90.26, 537.16, -5) mm, rotated rx -180 ry 0 rz 0 deg; joints [40.592, -49.392, 113.824, 43.799, -70.038, -17.11]
  MoveL 1569 to (64.86, 537.16, -5) mm, rotated rx -180 ry 0 rz 0 deg; joints [39.92, -48.582, 112.136, 43.339, -69.199, -17.527]
  MoveC 1570 to (61.14, 528.18, -5) mm, rotated rx -180 ry 0 rz 0 deg; joints [39.541, -48.694, 112.388, 42.918, -69.186, -17.294] to (52.16, 524.46, -5) mm, rotated rx -180 ry 0 rz 0 deg; joints [39.192, -48.498, 111.986, 42.615, -68.93, -17.321]
  MoveL 1571 to (52.16, 524.46, -5) mm, rotated rx -180 ry 0 rz 0 deg; joints [39.192, -48.498, 111.986, 42.615, -68.93, -17.321]
  MoveC 1572 to (43.18, 528.18, -5) mm, rotated rx -180 ry 0 rz 0 deg; joints [39.079, -48.108, 111.168, 42.612, -68.58, -17.592] to (39.46, 537.16, -5) mm, rotated rx 180 ry 0 rz 0 deg; joints [39.265, -47.752, 110.411, 42.91, -68.343, -17.952]
  MoveL 1573 to (14.06, 537.16, -5) mm, rotated rx -180 ry 0 rz 0 deg; joints [38.629, -46.904, 108.648, 42.51, -67.47, -18.386]
  MoveL 1574 to (14.06, 384.76, -5) mm, rotated rx -180 ry 0 rz 0 deg; joints [33.595, -50.528, 116.493, 36.247, -69.323, -13.664]
  MoveL 1575 to (19.05, 384.76, -5) mm, rotated rx -180 ry 0 rz 0 deg; joints [33.711, -50.696, 116.846, 36.328, -69.5, -13.588]
  MoveC 1576 to (19.49, 384.57, -5) mm, rotated rx -180 ry 0 rz 0 deg; joints [33.715, -50.715, 116.887, 36.327, -69.518, -13.576] to (19.68, 384.12, -5) mm, rotated rx -180 ry 0 rz 0 deg; joints [33.704, -50.731, 116.921, 36.311, -69.53, -13.56]
  MoveL 1577 to (19.68, 383.49, -5) mm, rotated rx 180 ry 0 rz 0 deg; joints [33.682, -50.744, 116.951, 36.284, -69.538, -13.542]
  MoveC 1578 to (19.68, 383.04, -4.81) mm, rotated rx 180 ry 0 rz 0 deg; joints [33.666, -50.765, 116.972, 36.268, -69.535, -13.536] to (19.68, 382.85, -4.37) mm, rotated rx 180 ry 0 rz 0 deg; joints [33.659, -50.795, 116.982, 36.265, -69.517, -13.547]
  Set speed (500.0 mm/s)
  MoveL 1579 to (19.68, 382.85, 5) mm, rotated rx -180 ry 0 rz 0 deg; joints [33.654, -51.338, 116.996, 36.378, -69.09, -13.88]
  MoveL 1580 to (18.41, 382.85, 5) mm, rotated rx -180 ry 0 rz 0 deg; joints [33.624, -51.294, 116.907, 36.358, -69.046, -13.898]
  Set speed (25.4 mm/s)
  MoveL 1581 to (18.41, 382.85, 1) mm, rotated rx -180 ry 0 rz 0 deg; joints [33.626, -51.063, 116.901, 36.309, -69.228, -13.756]
  MoveL 1582 to (18.41, 382.85, -7.72) mm, rotated rx 180 ry 0 rz 0 deg; joints [33.631, -50.558, 116.885, 36.205, -69.624, -13.448]
  MoveC 1583 to (18.41, 383.04, -8.16) mm, rotated rx -180 ry 0 rz 0 deg; joints [33.638, -50.527, 116.875, 36.207, -69.642, -13.438] to (18.41, 383.49, -8.35) mm, rotated rx -180 ry 0 rz 0 deg; joints [33.653, -50.507, 116.854, 36.224, -69.645, -13.444]
  Set speed (50.8 mm/s)
  MoveL 1584 to (18.41, 384.12, -8.35) mm, rotated rx -180 ry 0 rz 0 deg; joints [33.676, -50.493, 116.824, 36.251, -69.637, -13.462]
  MoveC 1585 to (18.6, 384.57, -8.35) mm, rotated rx 180 ry 0 rz 0 deg; joints [33.696, -50.49, 116.816, 36.273, -69.638, -13.472] to (19.04, 384.76, -8.35) mm, rotated rx 180 ry 0 rz 0 deg; joints [33.713, -50.501, 116.839, 36.288, -69.652, -13.47]
  MoveL 1586 to (64.86, 384.76, -8.35) mm, rotated rx 180 ry 0 rz 0 deg; joints [34.821, -52.002, 120.018, 37.076, -71.255, -12.772]
  MoveL 1587 to (471.26, 384.76, -8.35) mm, rotated rx -180 ry 0 rz 0 deg; joints [48.126, -62.955, 143.942, 48.578, -83.134, -6.474]
  MoveL 1588 to (471.26, 537.16, -8.35) mm, rotated rx 180 ry 0 rz 0 deg; joints [53.308, -59.215, 135.055, 54.322, -80.742, -11.191]
  MoveL 1589 to (445.86, 537.16, -8.35) mm, rotated rx -180 ry 0 rz 0 deg; joints [52.286, -58.665, 133.872, 53.393, -80.162, -11.557]
  MoveC 1590 to (433.16, 524.46, -8.35) mm, rotated rx -180 ry 0 rz 0 deg; joints [51.39, -58.719, 134.036, 52.487, -80.047, -11.328] to (420.46, 537.16, -8.35) mm, rotated rx -180 ry 0 rz 0 deg; joints [51.291, -58.099, 132.655, 52.498, -79.563, -11.925]
  MoveL 1591 to (395.06, 537.16, -8.35) mm, rotated rx 180 ry 0 rz 0 deg; joints [50.324, -57.516, 131.405, 51.635, -78.945, -12.296]
  MoveL 1592 to (318.86, 537.16, -8.35) mm, rotated rx -180 ry 0 rz 0 deg; joints [47.576, -55.667, 127.455, 49.245, -76.983, -13.424]
  MoveC 1593 to (306.16, 524.46, -8.35) mm, rotated rx -180 ry 0 rz 0 deg; joints [46.736, -55.674, 127.508, 48.398, -76.816, -13.211] to (293.46, 537.16, -8.35) mm, rotated rx -180 ry 0 rz 0 deg; joints [46.711, -55.017, 126.073, 48.513, -76.293, -13.804]
  MoveL 1594 to (191.86, 537.16, -8.35) mm, rotated rx -180 ry 0 rz 0 deg; joints [43.481, -52.249, 120.215, 45.892, -73.365, -15.357]
  MoveC 1595 to (179.16, 524.46, -8.35) mm, rotated rx -180 ry 0 rz 0 deg; joints [42.698, -52.211, 120.164, 45.107, -73.147, -15.151] to (166.46, 537.16, -8.35) mm, rotated rx -180 ry 0 rz 0 deg; joints [42.729, -51.514, 118.667, 45.313, -72.591, -15.754]
  MoveL 1596 to (90.26, 537.16, -8.35) mm, rotated rx -180 ry 0 rz 0 deg; joints [40.594, -49.204, 113.817, 43.755, -70.17, -16.977]
  MoveL 1597 to (64.86, 537.16, -8.35) mm, rotated rx 180 ry 0 rz 0 deg; joints [39.921, -48.397, 112.129, 43.295, -69.329, -17.397]
  MoveC 1598 to (61.14, 528.18, -8.35) mm, rotated rx 180 ry 0 rz 0 deg; joints [39.543, -48.509, 112.381, 42.873, -69.317, -17.165] to (52.16, 524.46, -8.35) mm, rotated rx -180 ry 0 rz 0 deg; joints [39.194, -48.313, 111.98, 42.57, -69.061, -17.193]
  MoveL 1599 to (52.16, 524.46, -8.35) mm, rotated rx -180 ry 0 rz 0 deg; joints [39.194, -48.313, 111.98, 42.57, -69.061, -17.193]
  MoveC 1600 to (43.18, 528.18, -8.35) mm, rotated rx -180 ry 0 rz 0 deg; joints [39.081, -47.925, 111.161, 42.568, -68.71, -17.465] to (39.46, 537.16, -8.35) mm, rotated rx -180 ry 0 rz 0 deg; joints [39.267, -47.571, 110.405, 42.864, -68.471, -17.825]
  MoveL 1601 to (14.06, 537.16, -8.35) mm, rotated rx -180 ry 0 rz 0 deg; joints [38.63, -46.725, 108.642, 42.464, -67.597, -18.261]
  MoveL 1602 to (14.06, 384.76, -8.35) mm, rotated rx -180 ry 0 rz 0 deg; joints [33.596, -50.334, 116.486, 36.208, -69.474, -13.547]
  MoveL 1603 to (19.04, 384.76, -8.35) mm, rotated rx 180 ry 0 rz 0 deg; joints [33.713, -50.501, 116.839, 36.288, -69.652, -13.47]
  MoveC 1604 to (19.49, 384.57, -8.35) mm, rotated rx -180 ry 0 rz 0 deg; joints [33.717, -50.52, 116.879, 36.287, -69.67, -13.458] to (19.68, 384.12, -8.35) mm, rotated rx -180 ry 0 rz 0 deg; joints [33.706, -50.536, 116.914, 36.272, -69.682, -13.442]
  MoveL 1605 to (19.68, 383.49, -8.35) mm, rotated rx 180 ry 0 rz 0 deg; joints [33.683, -50.549, 116.944, 36.245, -69.69, -13.424]
  MoveC 1606 to (19.68, 383.04, -8.16) mm, rotated rx -180 ry 0 rz 0 deg; joints [33.667, -50.57, 116.965, 36.228, -69.687, -13.418] to (19.68, 382.85, -7.72) mm, rotated rx 180 ry 0 rz 0 deg; joints [33.661, -50.6, 116.975, 36.225, -69.669, -13.429]
  Set speed (500.0 mm/s)
  MoveL 1607 to (19.68, 382.85, 6) mm, rotated rx -180 ry 0 rz 0 deg; joints [33.653, -51.395, 116.997, 36.39, -69.045, -13.915]
  MoveL 1608 to (-12.15, 384.12, 6) mm, rotated rx -180 ry 0 rz 0 deg; joints [32.964, -50.27, 114.666, 35.954, -67.899, -14.428]
  Set speed (25.4 mm/s)
  MoveL 1609 to (-12.15, 384.12, -4.37) mm, rotated rx -180 ry 0 rz 0 deg; joints [32.97, -49.686, 114.65, 35.826, -68.361, -14.07]
  MoveC 1610 to (-12.34, 384.12, -4.81) mm, rotated rx -180 ry 0 rz 0 deg; joints [32.966, -49.654, 114.636, 35.817, -68.374, -14.058] to (-12.79, 384.12, -5) mm, rotated rx -180 ry 0 rz 0 deg; joints [32.955, -49.628, 114.603, 35.808, -68.366, -14.058]
  Set speed (50.8 mm/s)
  MoveL 1611 to (-13.42, 384.12, -5) mm, rotated rx -180 ry 0 rz 0 deg; joints [32.941, -49.606, 114.557, 35.799, -68.343, -14.068]
  MoveC 1612 to (-13.87, 384.31, -5) mm, rotated rx 180 ry 0 rz 0 deg; joints [32.937, -49.587, 114.516, 35.8, -68.325, -14.081] to (-14.06, 384.76, -5) mm, rotated rx -180 ry 0 rz 0 deg; joints [32.949, -49.57, 114.482, 35.816, -68.313, -14.096]
  MoveL 1613 to (-14.06, 537.16, -5) mm, rotated rx 180 ry 0 rz 0 deg; joints [37.944, -45.941, 106.651, 42.102, -66.483, -18.877]
  MoveL 1614 to (-39.46, 537.16, -5) mm, rotated rx -180 ry 0 rz 0 deg; joints [37.343, -45.049, 104.803, 41.766, -65.573, -19.334]
  MoveC 1615 to (-52.16, 524.46, -5) mm, rotated rx -180 ry 0 rz 0 deg; joints [36.659, -44.926, 104.571, 41.09, -65.262, -19.129] to (-64.86, 537.16, -5) mm, rotated rx -180 ry 0 rz 0 deg; joints [36.758, -44.135, 102.913, 41.46, -64.644, -19.802]
  MoveL 1616 to (-90.26, 537.16, -5) mm, rotated rx 180 ry 0 rz 0 deg; joints [36.189, -43.198, 100.977, 41.186, -63.696, -20.285]
  MoveL 1617 to (-166.46, 537.16, -5) mm, rotated rx -180 ry 0 rz 0 deg; joints [34.57, -40.24, 94.878, 40.564, -60.732, -21.838]
  MoveC 1618 to (-179.16, 524.46, -5) mm, rotated rx -180 ry 0 rz 0 deg; joints [33.935, -40.066, 94.539, 39.949, -60.368, -21.638] to (-191.86, 537.16, -5) mm, rotated rx -180 ry 0 rz 0 deg; joints [34.058, -39.2, 92.738, 40.427, -59.701, -22.398]
  MoveL 1619 to (-293.46, 537.16, -5) mm, rotated rx -180 ry 0 rz 0 deg; joints [32.138, -34.713, 83.533, 40.292, -55.325, -24.932]
  MoveC 1620 to (-306.16, 524.46, -5) mm, rotated rx -180 ry 0 rz 0 deg; joints [31.548, -34.478, 83.066, 39.746, -54.897, -24.75] to (-318.86, 537.16, -5) mm, rotated rx -180 ry 0 rz 0 deg; joints [31.687, -33.497, 81.042, 40.378, -54.159, -25.662]
  MoveL 1621 to (-395.06, 537.16, -5) mm, rotated rx 180 ry 0 rz 0 deg; joints [30.402, -29.552, 72.982, 41.008, -50.451, -28.189]
  MoveL 1622 to (-420.46, 537.16, -5) mm, rotated rx 180 ry 0 rz 0 deg; joints [29.995, -28.119, 70.057, 41.371, -49.131, -29.18]
  MoveC 1623 to (-433.16, 524.46, -5) mm, rotated rx -180 ry 0 rz 0 deg; joints [29.446, -27.794, 69.409, 40.922, -48.618, -29.053] to (-445.86, 537.16, -5) mm, rotated rx -180 ry 0 rz 0 deg; joints [29.597, -26.611, 66.985, 41.832, -47.762, -30.269]
  MoveL 1624 to (-471.26, 537.16, -5) mm, rotated rx -180 ry 0 rz 0 deg; joints [29.209, -25.018, 63.739, 42.41, -46.335, -31.48]
  MoveL 1625 to (-471.26, 384.76, -5) mm, rotated rx 180 ry 0 rz 0 deg; joints [24.926, -29.68, 73.401, 34.382, -48.254, -23.818]
  MoveL 1626 to (-14.06, 384.76, -5) mm, rotated rx -180 ry 0 rz 0 deg; joints [32.949, -49.57, 114.482, 35.816, -68.313, -14.096]
  MoveC 1627 to (-13.61, 384.57, -5) mm, rotated rx 180 ry 0 rz 0 deg; joints [32.953, -49.59, 114.523, 35.815, -68.331, -14.084] to (-13.42, 384.12, -5) mm, rotated rx -180 ry 0 rz 0 deg; joints [32.941, -49.606, 114.557, 35.799, -68.343, -14.068]
  MoveL 1628 to (-13.42, 383.49, -5) mm, rotated rx 180 ry 0 rz 0 deg; joints [32.919, -49.62, 114.587, 35.772, -68.351, -14.05]
  MoveC 1629 to (-13.42, 383.04, -4.81) mm, rotated rx -180 ry 0 rz 0 deg; joints [32.903, -49.64, 114.608, 35.756, -68.348, -14.043] to (-13.42, 382.85, -4.37) mm, rotated rx -180 ry 0 rz 0 deg; joints [32.897, -49.669, 114.618, 35.753, -68.33, -14.053]
  Set speed (500.0 mm/s)
  MoveL 1630 to (-13.42, 382.85, 5) mm, rotated rx -180 ry 0 rz 0 deg; joints [32.892, -50.197, 114.632, 35.869, -67.912, -14.376]
  MoveL 1631 to (-12.15, 384.12, 5) mm, rotated rx -180 ry 0 rz 0 deg; joints [32.965, -50.214, 114.665, 35.941, -67.944, -14.393]
  Set speed (25.4 mm/s)
  MoveL 1632 to (-12.15, 384.12, 1) mm, rotated rx -180 ry 0 rz 0 deg; joints [32.967, -49.989, 114.659, 35.891, -68.122, -14.255]
  MoveL 1633 to (-12.15, 384.12, -7.72) mm, rotated rx -180 ry 0 rz 0 deg; joints [32.971, -49.496, 114.643, 35.785, -68.51, -13.956]
  MoveC 1634 to (-12.34, 384.12, -8.16) mm, rotated rx -180 ry 0 rz 0 deg; joints [32.967, -49.464, 114.629, 35.777, -68.523, -13.944] to (-12.79, 384.12, -8.35) mm, rotated rx 180 ry 0 rz 0 deg; joints [32.957, -49.438, 114.596, 35.768, -68.515, -13.944]
  Set speed (50.8 mm/s)
  MoveL 1635 to (-13.42, 384.12, -8.35) mm, rotated rx 180 ry 0 rz 0 deg; joints [32.943, -49.416, 114.55, 35.759, -68.492, -13.954]
  MoveC 1636 to (-13.87, 384.31, -8.35) mm, rotated rx 180 ry 0 rz 0 deg; joints [32.939, -49.397, 114.509, 35.76, -68.473, -13.966] to (-14.06, 384.76, -8.35) mm, rotated rx 180 ry 0 rz 0 deg; joints [32.951, -49.381, 114.475, 35.776, -68.461, -13.982]
  MoveL 1637 to (-14.06, 537.16, -8.35) mm, rotated rx 180 ry 0 rz 0 deg; joints [37.946, -45.766, 106.644, 42.055, -66.608, -18.755]
  MoveL 1638 to (-39.46, 537.16, -8.35) mm, rotated rx -180 ry 0 rz 0 deg; joints [37.345, -44.877, 104.796, 41.718, -65.696, -19.214]
  MoveC 1639 to (-52.16, 524.46, -8.35) mm, rotated rx -180 ry 0 rz 0 deg; joints [36.661, -44.755, 104.564, 41.042, -65.387, -19.011] to (-64.86, 537.16, -8.35) mm, rotated rx -180 ry 0 rz 0 deg; joints [36.76, -43.966, 102.906, 41.411, -64.766, -19.685]
  MoveL 1640 to (-90.26, 537.16, -8.35) mm, rotated rx -180 ry 0 rz 0 deg; joints [36.191, -43.032, 100.97, 41.136, -63.816, -20.169]
  MoveL 1641 to (-166.46, 537.16, -8.35) mm, rotated rx 180 ry 0 rz 0 deg; joints [34.571, -40.082, 94.872, 40.511, -60.847, -21.726]
  MoveC 1642 to (-179.16, 524.46, -8.35) mm, rotated rx 180 ry 0 rz 0 deg; joints [33.937, -39.909, 94.532, 39.896, -60.484, -21.528] to (-191.86, 537.16, -8.35) mm, rotated rx 180 ry 0 rz 0 deg; joints [34.059, -39.044, 92.731, 40.373, -59.814, -22.287]
  MoveL 1643 to (-293.46, 537.16, -8.35) mm, rotated rx 180 ry 0 rz 0 deg; joints [32.139, -34.568, 83.526, 40.232, -55.431, -24.824]
  MoveC 1644 to (-306.16, 524.46, -8.35) mm, rotated rx -180 ry 0 rz 0 deg; joints [31.549, -34.332, 83.059, 39.685, -55.004, -24.643] to (-318.86, 537.16, -8.35) mm, rotated rx -180 ry 0 rz 0 deg; joints [31.689, -33.353, 81.035, 40.316, -54.264, -25.554]
  MoveL 1645 to (-395.06, 537.16, -8.35) mm, rotated rx 180 ry 0 rz 0 deg; joints [30.404, -29.415, 72.974, 40.939, -50.549, -28.08]
  MoveL 1646 to (-420.46, 537.16, -8.35) mm, rotated rx 180 ry 0 rz 0 deg; joints [29.996, -27.983, 70.049, 41.3, -49.228, -29.069]
  MoveC 1647 to (-433.16, 524.46, -8.35) mm, rotated rx 180 ry 0 rz 0 deg; joints [29.447, -27.659, 69.401, 40.85, -48.715, -28.943] to (-445.86, 537.16, -8.35) mm, rotated rx -180 ry 0 rz 0 deg; joints [29.598, -26.477, 66.976, 41.758, -47.856, -30.157]
  MoveL 1648 to (-471.26, 537.16, -8.35) mm, rotated rx -180 ry 0 rz 0 deg; joints [29.21, -24.886, 63.73, 42.332, -46.427, -31.366]
  MoveL 1649 to (-471.26, 384.76, -8.35) mm, rotated rx 180 ry 0 rz 0 deg; joints [24.927, -29.542, 73.394, 34.319, -48.362, -23.72]
  MoveL 1650 to (-14.06, 384.76, -8.35) mm, rotated rx -180 ry 0 rz 0 deg; joints [32.951, -49.381, 114.475, 35.776, -68.461, -13.982]
  MoveC 1651 to (-13.61, 384.57, -8.35) mm, rotated rx -180 ry 0 rz 0 deg; joints [32.954, -49.4, 114.516, 35.775, -68.48, -13.97] to (-13.42, 384.12, -8.35) mm, rotated rx 180 ry 0 rz 0 deg; joints [32.943, -49.416, 114.55, 35.759, -68.492, -13.954]
  MoveL 1652 to (-13.42, 383.49, -8.35) mm, rotated rx -180 ry 0 rz 0 deg; joints [32.921, -49.43, 114.58, 35.732, -68.5, -13.936]
  MoveC 1653 to (-13.42, 383.04, -8.16) mm, rotated rx -180 ry 0 rz 0 deg; joints [32.905, -49.45, 114.601, 35.715, -68.497, -13.929] to (-13.42, 382.85, -7.72) mm, rotated rx -180 ry 0 rz 0 deg; joints [32.898, -49.479, 114.611, 35.713, -68.479, -13.939]
  Set speed (500.0 mm/s)
  MoveL 1654 to (-13.42, 382.85, 15) mm, rotated rx 180 ry 0 rz 0 deg; joints [32.887, -50.758, 114.64, 35.997, -67.463, -14.725]
  MoveL 1655 to (-13.42, 382.85, 15) mm, rotated rx 180 ry 0 rz 0 deg; joints [32.887, -50.758, 114.64, 35.997, -67.463, -14.725]

--- program Prog2 (robot GIGASHEEN) ---
  MoveJ (plywood back right safe) [its target is no longer in the station]
  MoveL (plywood back left safe) [its target is no longer in the station]
  MoveL (plywood front left safe) [its target is no longer in the station]
  MoveL (plywood front right safe) [its target is no longer in the station]
